LIN {X 0,Y 303.642,Z 314.333,A -85,B 0,C 180,E1 -15935.578,E2 -15935.578} C_VEL
LIN {X 0,Y 303.878,Z 309.685,A -85,B 0,C 180,E1 -15937.976,E2 -15937.976} C_VEL
LIN {X 0,Y 304.337,Z 303.514,A -85,B 0,C 180,E1 -15940.309,E2 -15940.309} C_VEL
LIN {X 0,Y 305.034,Z 296.766,A -85,B 0,C 180,E1 -15942.305,E2 -15942.305} C_VEL
LIN {X 0,Y 306.049,Z 288.388,A -85,B 0,C 180,E1 -15944.291,E2 -15944.291} C_VEL
LIN {X 0,Y 307.158,Z 279.773,A -85,B 0,C 180,E1 -15945.936,E2 -15945.936} C_VEL
LIN {X 0,Y 308.289,Z 269.101,A -85,B 0,C 180,E1 -15947.581,E2 -15947.581} C_VEL
LIN {X 0,Y 309.733,Z 258.568,A -85,B 0,C 180,E1 -15948.865,E2 -15948.865} C_VEL
LIN {X 0,Y 310.948,Z 246.911,A -85,B 0,C 180,E1 -15949.989,E2 -15949.989} C_VEL
LIN {X 0,Y 312.046,Z 234.79,A -85,B 0,C 180,E1 -15950.863,E2 -15950.863} C_VEL
LIN {X 0,Y 313.009,Z 221.635,A -85,B 0,C 180,E1 -15951.528,E2 -15951.528} C_VEL
LIN {X 0,Y 313.468,Z 208.98,A -85,B 0,C 180,E1 -15951.927,E2 -15951.927} C_VEL
LIN {X 0,Y 314.607,Z 149.7,A -85,B 0,C 180,E1 -15953.265,E2 -15953.265} C_VEL
LIN {X 0,Y 309.854,Z 113.898,A -85,B 0,C 180,E1 -15954.459,E2 -15954.459} C_VEL
LIN {X 0,Y 308.762,Z 106.65,A -85,B 0,C 180,E1 -15954.726,E2 -15954.726} C_VEL
LIN {X 0,Y 309.513,Z 100.612,A -85,B 0,C 180,E1 -15956.281,E2 -15956.281} C_VEL
LIN {X 0,Y 308.694,Z 94.627,A -85,B 0,C 180,E1 -15957.946,E2 -15957.946} C_VEL
LIN {X 0,Y 306.773,Z 85.34,A -85,B 0,C 180,E1 -15960.646,E2 -15960.646} C_VEL
LIN {X 0,Y 305.49,Z 79.435,A -85,B 0,C 180,E1 -15962.433,E2 -15962.433} C_VEL
LIN {X 0,Y 305.496,Z 79.432,A -85,B 0,C 180,E1 -15966.736,E2 -15966.736} C_VEL
LIN {X 0,Y 305.454,Z 79.435,A -85,B 0,C 180,E1 -15970.6,E2 -15970.6} C_VEL
LIN {X 0,Y 305.424,Z 79.442,A -85,B 0,C 180,E1 -15973.655,E2 -15973.655} C_VEL
LIN {X 0,Y 305.454,Z 79.438,A -85,B 0,C 180,E1 -15977.414,E2 -15977.414} C_VEL
LIN {X 0,Y 305.475,Z 79.428,A -85,B 0,C 180,E1 -15981.597,E2 -15981.597} C_VEL
LIN {X 0,Y 305.461,Z 79.435,A -85,B 0,C 180,E1 -15984.887,E2 -15984.887} C_VEL
LIN {X 0,Y 305.451,Z 79.435,A -85,B 0,C 180,E1 -15988.355,E2 -15988.355} C_VEL
LIN {X 0,Y 305.519,Z 79.429,A -85,B 0,C 180,E1 -15991.114,E2 -15991.114} C_VEL
LIN {X 0,Y 305.57,Z 79.417,A -85,B 0,C 180,E1 -15994.088,E2 -15994.088} C_VEL
LIN {X 0,Y 305.5,Z 79.429,A -85,B 0,C 180,E1 -15998.403,E2 -15998.403} C_VEL
LIN {X 0,Y 305.589,Z 79.417,A -85,B 0,C 180,E1 -16001.218,E2 -16001.218} C_VEL
LIN {X 0,Y 305.648,Z 79.408,A -85,B 0,C 180,E1 -16005.349,E2 -16005.349} C_VEL
LIN {X 0,Y 305.635,Z 79.409,A -85,B 0,C 180,E1 -16009.4,E2 -16009.4} C_VEL
LIN {X 0,Y 305.796,Z 79.394,A -85,B 0,C 180,E1 -16012.074,E2 -16012.074} C_VEL
LIN {X 0,Y 305.682,Z 79.404,A -85,B 0,C 180,E1 -16014.724,E2 -16014.724} C_VEL
LIN {X 0,Y 305.953,Z 79.372,A -85,B 0,C 180,E1 -16018.684,E2 -16018.684} C_VEL
LIN {X 0,Y 305.953,Z 79.372,A -85,B 0,C 180,E1 -16021.317,E2 -16021.317} C_VEL
LIN {X 0,Y 305.672,Z 79.402,A -85,B 0,C 180,E1 -16025.277,E2 -16025.277} C_VEL
LIN {X 0,Y 305.764,Z 79.399,A -85,B 0,C 180,E1 -16027.927,E2 -16027.927} C_VEL
LIN {X 0,Y 305.598,Z 79.414,A -85,B 0,C 180,E1 -16031.946,E2 -16031.946} C_VEL
LIN {X 0,Y 305.637,Z 79.409,A -85,B 0,C 180,E1 -16035.035,E2 -16035.035} C_VEL
LIN {X 0,Y 305.576,Z 79.42,A -85,B 0,C 180,E1 -16039.445,E2 -16039.445} C_VEL
LIN {X 0,Y 305.491,Z 79.428,A -85,B 0,C 180,E1 -16043.042,E2 -16043.042} C_VEL
LIN {X 0,Y 305.526,Z 79.424,A -85,B 0,C 180,E1 -16046.219,E2 -16046.219} C_VEL
LIN {X 0,Y 305.489,Z 79.433,A -85,B 0,C 180,E1 -16049.048,E2 -16049.048} C_VEL
LIN {X 0,Y 305.442,Z 79.435,A -85,B 0,C 180,E1 -16051.953,E2 -16051.953} C_VEL
LIN {X 0,Y 305.462,Z 79.437,A -85,B 0,C 180,E1 -16055.114,E2 -16055.114} C_VEL
LIN {X 0,Y 305.434,Z 79.438,A -85,B 0,C 180,E1 -16058.526,E2 -16058.526} C_VEL
LIN {X 0,Y 305.436,Z 79.44,A -85,B 0,C 180,E1 -16062.582,E2 -16062.582} C_VEL
LIN {X 0,Y 305.424,Z 79.441,A -85,B 0,C 180,E1 -16066.345,E2 -16066.345} C_VEL
LIN {X 0,Y 305.459,Z 79.434,A -85,B 0,C 180,E1 -16069.893,E2 -16069.893} C_VEL
LIN {X 0,Y 305.465,Z 79.433,A -85,B 0,C 180,E1 -16073.637,E2 -16073.637} C_VEL
LIN {X 0,Y 305.467,Z 79.434,A -85,B 0,C 180,E1 -16076.484,E2 -16076.484} C_VEL
LIN {X 0,Y 305.433,Z 79.437,A -85,B 0,C 180,E1 -16079.588,E2 -16079.588} C_VEL
LIN {X 0,Y 305.455,Z 79.436,A -85,B 0,C 180,E1 -16082.603,E2 -16082.603} C_VEL
LIN {X 0,Y 305.461,Z 79.435,A -85,B 0,C 180,E1 -16085.535,E2 -16085.535} C_VEL
LIN {X 0,Y 305.515,Z 79.431,A -85,B 0,C 180,E1 -16089.815,E2 -16089.815} C_VEL
LIN {X 0,Y 305.651,Z 79.555,A -85,B 0,C 180,E1 -16091.396,E2 -16091.396} C_VEL
LIN {X 0,Y 306.172,Z 82.09,A -85,B 0,C 180,E1 -16092.18,E2 -16092.18} C_VEL
LIN {X 0,Y 314.171,Z 104.116,A -85,B 0,C 180,E1 -16093.31,E2 -16093.31} C_VEL
LIN {X 0,Y 315.408,Z 109.173,A -85,B 0,C 180,E1 -16093.518,E2 -16093.518} C_VEL
LIN {X 0,Y 313.679,Z 189.055,A -85,B 0,C 180,E1 -16095.346,E2 -16095.346} C_VEL
LIN {X 0,Y 313.088,Z 202.338,A -85,B 0,C 180,E1 -16095.912,E2 -16095.912} C_VEL
LIN {X 0,Y 312.343,Z 214.286,A -85,B 0,C 180,E1 -16096.666,E2 -16096.666} C_VEL
LIN {X 0,Y 311.528,Z 225.57,A -85,B 0,C 180,E1 -16097.625,E2 -16097.625} C_VEL
LIN {X 0,Y 310.283,Z 237.207,A -85,B 0,C 180,E1 -16098.9,E2 -16098.9} C_VEL
LIN {X 0,Y 309.036,Z 247.649,A -85,B 0,C 180,E1 -16100.345,E2 -16100.345} C_VEL
LIN {X 0,Y 307.882,Z 256.196,A -85,B 0,C 180,E1 -16101.798,E2 -16101.798} C_VEL
LIN {X 0,Y 306.867,Z 264.064,A -85,B 0,C 180,E1 -16103.425,E2 -16103.425} C_VEL
LIN {X 0,Y 305.788,Z 271.78,A -85,B 0,C 180,E1 -16105.386,E2 -16105.386} C_VEL
LIN {X 0,Y 305.065,Z 277.948,A -85,B 0,C 180,E1 -16107.36,E2 -16107.36} C_VEL
LIN {X 0,Y 304.464,Z 282.865,A -85,B 0,C 180,E1 -16109.339,E2 -16109.339} C_VEL
LIN {X 0,Y 304.148,Z 286.666,A -85,B 0,C 180,E1 -16111.324,E2 -16111.324} C_VEL
LIN {X 0,Y 303.886,Z 288.636,A -85,B 0,C 180,E1 -16112.652,E2 -16112.652} C_VEL
LIN {X 0,Y 303.852,Z 290.188,A -85,B 0,C 180,E1 -16113.979,E2 -16113.979} C_VEL
LIN {X 0,Y 303.867,Z 291.727,A -85,B 0,C 180,E1 -16115.991,E2 -16115.991} C_VEL
LIN {X 0,Y 303.757,Z 292.363,A -85,B 0,C 180,E1 -16117.98,E2 -16117.98} C_VEL
LIN {X 0,Y 303.781,Z 292.317,A -85,B 0,C 180,E1 -16119.32,E2 -16119.32} C_VEL
LIN {X 0,Y 303.861,Z 291.854,A -85,B 0,C 180,E1 -16120.663,E2 -16120.663} C_VEL
LIN {X 0,Y 304.117,Z 290.967,A -85,B 0,C 180,E1 -16122.005,E2 -16122.005} C_VEL
LIN {X 0,Y 304.786,Z 288.35,A -85,B 0,C 180,E1 -16124.423,E2 -16124.423} C_VEL
LIN {X 0,Y 305.573,Z 284.582,A -85,B 0,C 180,E1 -16126.708,E2 -16126.708} C_VEL
LIN {X 0,Y 306.602,Z 280.053,A -85,B 0,C 180,E1 -16128.718,E2 -16128.718} C_VEL
LIN {X 0,Y 307.928,Z 273.826,A -85,B 0,C 180,E1 -16130.852,E2 -16130.852} C_VEL
LIN {X 0,Y 309.428,Z 266.966,A -85,B 0,C 180,E1 -16132.714,E2 -16132.714} C_VEL
LIN {X 0,Y 311.294,Z 257.875,A -85,B 0,C 180,E1 -16134.688,E2 -16134.688} C_VEL
LIN {X 0,Y 313.036,Z 248.077,A -85,B 0,C 180,E1 -16136.376,E2 -16136.376} C_VEL
LIN {X 0,Y 314.749,Z 237.818,A -85,B 0,C 180,E1 -16137.783,E2 -16137.783} C_VEL
LIN {X 0,Y 316.501,Z 225.991,A -85,B 0,C 180,E1 -16139.062,E2 -16139.062} C_VEL
LIN {X 0,Y 317.895,Z 214.405,A -85,B 0,C 180,E1 -16140.013,E2 -16140.013} C_VEL
LIN {X 0,Y 318.974,Z 201.792,A -85,B 0,C 180,E1 -16140.782,E2 -16140.782} C_VEL
LIN {X 0,Y 319.8,Z 188.955,A -85,B 0,C 180,E1 -16141.299,E2 -16141.299} C_VEL
LIN {X 0,Y 321.712,Z 116.244,A -85,B 0,C 180,E1 -16142.959,E2 -16142.959} C_VEL
LIN {X 0,Y 314.092,Z 98.688,A -85,B 0,C 180,E1 -16144.191,E2 -16144.191} C_VEL
LIN {X 0,Y 307.154,Z 84.745,A -85,B 0,C 180,E1 -16145.326,E2 -16145.326} C_VEL
LIN {X 0,Y 306.212,Z 82.518,A -85,B 0,C 180,E1 -16145.534,E2 -16145.534} C_VEL
LIN {X 0,Y 305.477,Z 79.43,A -85,B 0,C 180,E1 -16146.74,E2 -16146.74} C_VEL
LIN {X 0,Y 305.438,Z 79.432,A -85,B 0,C 180,E1 -16147.526,E2 -16147.526} C_VEL
LIN {X 0,Y 304.776,Z 79.521,A -85,B 0,C 180,E1 -16148.626,E2 -16148.626} C_VEL
LIN {X 0,Y 301.946,Z 79.88,A -85,B 0,C 180,E1 -16150.419,E2 -16150.419} C_VEL
LIN {X 0,Y 299.525,Z 80.183,A -85,B 0,C 180,E1 -16151.872,E2 -16151.872} C_VEL
LIN {X 0,Y 298.454,Z 80.309,A -85,B 0,C 180,E1 -16152.998,E2 -16152.998} C_VEL
LIN {X 0,Y 298.351,Z 80.315,A -85,B 0,C 180,E1 -16153.379,E2 -16153.379} C_VEL
LIN {X 0,Y 298.373,Z 80.318,A -85,B 0,C 180,E1 -16156.915,E2 -16156.915} C_VEL
LIN {X 0,Y 298.388,Z 80.313,A -85,B 0,C 180,E1 -16161.011,E2 -16161.011} C_VEL
LIN {X 0,Y 298.407,Z 80.31,A -85,B 0,C 180,E1 -16163.928,E2 -16163.928} C_VEL
LIN {X 0,Y 298.395,Z 80.314,A -85,B 0,C 180,E1 -16167.199,E2 -16167.199} C_VEL
LIN {X 0,Y 298.409,Z 80.307,A -85,B 0,C 180,E1 -16171.898,E2 -16171.898} C_VEL
LIN {X 0,Y 298.441,Z 80.312,A -85,B 0,C 180,E1 -16174.92,E2 -16174.92} C_VEL
LIN {X 0,Y 298.407,Z 80.305,A -85,B 0,C 180,E1 -16177.862,E2 -16177.862} C_VEL
LIN {X 0,Y 298.511,Z 80.298,A -85,B 0,C 180,E1 -16180.755,E2 -16180.755} C_VEL
LIN {X 0,Y 298.589,Z 80.293,A -85,B 0,C 180,E1 -16184.994,E2 -16184.994} C_VEL
LIN {X 0,Y 298.586,Z 80.285,A -85,B 0,C 180,E1 -16189.146,E2 -16189.146} C_VEL
LIN {X 0,Y 298.7,Z 80.277,A -85,B 0,C 180,E1 -16191.884,E2 -16191.884} C_VEL
LIN {X 0,Y 298.633,Z 80.274,A -85,B 0,C 180,E1 -16194.598,E2 -16194.598} C_VEL
LIN {X 0,Y 298.907,Z 80.242,A -85,B 0,C 180,E1 -16198.652,E2 -16198.652} C_VEL
LIN {X 0,Y 298.916,Z 80.244,A -85,B 0,C 180,E1 -16201.347,E2 -16201.347} C_VEL
LIN {X 0,Y 298.738,Z 80.261,A -85,B 0,C 180,E1 -16206.755,E2 -16206.755} C_VEL
LIN {X 0,Y 298.629,Z 80.286,A -85,B 0,C 180,E1 -16209.482,E2 -16209.482} C_VEL
LIN {X 0,Y 298.548,Z 80.292,A -85,B 0,C 180,E1 -16213.615,E2 -16213.615} C_VEL
LIN {X 0,Y 298.489,Z 80.293,A -85,B 0,C 180,E1 -16216.412,E2 -16216.412} C_VEL
LIN {X 0,Y 298.501,Z 80.303,A -85,B 0,C 180,E1 -16219.647,E2 -16219.647} C_VEL
LIN {X 0,Y 298.46,Z 80.304,A -85,B 0,C 180,E1 -16223.597,E2 -16223.597} C_VEL
LIN {X 0,Y 298.492,Z 80.295,A -85,B 0,C 180,E1 -16226.574,E2 -16226.574} C_VEL
LIN {X 0,Y 298.419,Z 80.311,A -85,B 0,C 180,E1 -16229.641,E2 -16229.641} C_VEL
LIN {X 0,Y 298.397,Z 80.316,A -85,B 0,C 180,E1 -16232.8,E2 -16232.8} C_VEL
LIN {X 0,Y 298.449,Z 80.281,A -85,B 0,C 180,E1 -16236.807,E2 -16236.807} C_VEL
LIN {X 0,Y 298.411,Z 80.314,A -85,B 0,C 180,E1 -16239.486,E2 -16239.486} C_VEL
LIN {X 0,Y 298.4,Z 80.315,A -85,B 0,C 180,E1 -16243.103,E2 -16243.103} C_VEL
LIN {X 0,Y 298.405,Z 80.312,A -85,B 0,C 180,E1 -16246.92,E2 -16246.92} C_VEL
LIN {X 0,Y 298.406,Z 80.311,A -85,B 0,C 180,E1 -16251.006,E2 -16251.006} C_VEL
LIN {X 0,Y 298.421,Z 80.369,A -85,B 0,C 180,E1 -16252.844,E2 -16252.844} C_VEL
LIN {X 0,Y 301.194,Z 91.103,A -85,B 0,C 180,E1 -16256.622,E2 -16256.622} C_VEL
LIN {X 0,Y 303.877,Z 103.194,A -85,B 0,C 180,E1 -16260.563,E2 -16260.563} C_VEL
LIN {X 0,Y 304.366,Z 105.671,A -85,B 0,C 180,E1 -16261.335,E2 -16261.335} C_VEL
LIN {X 0,Y 307.278,Z 113.342,A -85,B 0,C 180,E1 -16261.877,E2 -16261.877} C_VEL
LIN {X 0,Y 312.669,Z 141.354,A -85,B 0,C 180,E1 -16263.189,E2 -16263.189} C_VEL
LIN {X 0,Y 314.565,Z 154.061,A -85,B 0,C 180,E1 -16263.709,E2 -16263.709} C_VEL
LIN {X 0,Y 312.73,Z 215.019,A -85,B 0,C 180,E1 -16265.123,E2 -16265.123} C_VEL
LIN {X 0,Y 311.67,Z 228.866,A -85,B 0,C 180,E1 -16265.699,E2 -16265.699} C_VEL
LIN {X 0,Y 310.181,Z 241.295,A -85,B 0,C 180,E1 -16266.462,E2 -16266.462} C_VEL
LIN {X 0,Y 308.6,Z 252.386,A -85,B 0,C 180,E1 -16267.399,E2 -16267.399} C_VEL
LIN {X 0,Y 306.694,Z 263.941,A -85,B 0,C 180,E1 -16268.667,E2 -16268.667} C_VEL
LIN {X 0,Y 304.7,Z 274.36,A -85,B 0,C 180,E1 -16270.11,E2 -16270.11} C_VEL
LIN {X 0,Y 302.78,Z 283.763,A -85,B 0,C 180,E1 -16271.738,E2 -16271.738} C_VEL
LIN {X 0,Y 300.962,Z 292.85,A -85,B 0,C 180,E1 -16273.726,E2 -16273.726} C_VEL
LIN {X 0,Y 299.458,Z 300.197,A -85,B 0,C 180,E1 -16275.733,E2 -16275.733} C_VEL
LIN {X 0,Y 298.128,Z 306.106,A -85,B 0,C 180,E1 -16277.75,E2 -16277.75} C_VEL
LIN {X 0,Y 297.363,Z 310.791,A -85,B 0,C 180,E1 -16279.789,E2 -16279.789} C_VEL
LIN {X 0,Y 296.856,Z 314.38,A -85,B 0,C 180,E1 -16281.833,E2 -16281.833} C_VEL
LIN {X 0,Y 296.649,Z 316.232,A -85,B 0,C 180,E1 -16283.197,E2 -16283.197} C_VEL
LIN {X 0,Y 296.566,Z 318.639,A -85,B 0,C 180,E1 -16285.923,E2 -16285.923} C_VEL
LIN {X 0,Y 296.578,Z 319.259,A -85,B 0,C 180,E1 -16287.283,E2 -16287.283} C_VEL
LIN {X 0,Y 296.597,Z 319.477,A -85,B 0,C 180,E1 -16288.642,E2 -16288.642} C_VEL
LIN {X 0,Y 296.672,Z 319.265,A -85,B 0,C 180,E1 -16290,E2 -16290} C_VEL
LIN {X 0,Y 296.614,Z 318.655,A -85,B 0,C 180,E1 -16291.357,E2 -16291.357} C_VEL
LIN {X 0,Y 296.612,Z 317.653,A -85,B 0,C 180,E1 -16292.716,E2 -16292.716} C_VEL
LIN {X 0,Y 296.608,Z 316.234,A -85,B 0,C 180,E1 -16294.076,E2 -16294.076} C_VEL
LIN {X 0,Y 296.57,Z 313.254,A -85,B 0,C 180,E1 -16296.121,E2 -16296.121} C_VEL
LIN {X 0,Y 296.822,Z 309.219,A -85,B 0,C 180,E1 -16298.167,E2 -16298.167} C_VEL
LIN {X 0,Y 297.317,Z 302.992,A -85,B 0,C 180,E1 -16300.556,E2 -16300.556} C_VEL
LIN {X 0,Y 298.073,Z 296.199,A -85,B 0,C 180,E1 -16302.597,E2 -16302.597} C_VEL
LIN {X 0,Y 299.144,Z 287.762,A -85,B 0,C 180,E1 -16304.628,E2 -16304.628} C_VEL
LIN {X 0,Y 300.236,Z 279.054,A -85,B 0,C 180,E1 -16306.313,E2 -16306.313} C_VEL
LIN {X 0,Y 301.318,Z 269.493,A -85,B 0,C 180,E1 -16307.826,E2 -16307.826} C_VEL
LIN {X 0,Y 302.989,Z 257.676,A -85,B 0,C 180,E1 -16309.301,E2 -16309.301} C_VEL
LIN {X 0,Y 304.247,Z 245.794,A -85,B 0,C 180,E1 -16310.449,E2 -16310.449} C_VEL
LIN {X 0,Y 305.395,Z 233.429,A -85,B 0,C 180,E1 -16311.339,E2 -16311.339} C_VEL
LIN {X 0,Y 306.33,Z 220.772,A -85,B 0,C 180,E1 -16311.978,E2 -16311.978} C_VEL
LIN {X 0,Y 306.817,Z 207.603,A -85,B 0,C 180,E1 -16312.384,E2 -16312.384} C_VEL
LIN {X 0,Y 307.946,Z 150.508,A -85,B 0,C 180,E1 -16313.7,E2 -16313.7} C_VEL
LIN {X 0,Y 303.523,Z 116.739,A -85,B 0,C 180,E1 -16314.855,E2 -16314.855} C_VEL
LIN {X 0,Y 301.95,Z 106.265,A -85,B 0,C 180,E1 -16315.262,E2 -16315.262} C_VEL
LIN {X 0,Y 302.573,Z 101.353,A -85,B 0,C 180,E1 -16316.559,E2 -16316.559} C_VEL
LIN {X 0,Y 301.205,Z 93.039,A -85,B 0,C 180,E1 -16318.957,E2 -16318.957} C_VEL
LIN {X 0,Y 298.456,Z 80.312,A -85,B 0,C 180,E1 -16322.842,E2 -16322.842} C_VEL
LIN {X 0,Y 298.464,Z 80.309,A -85,B 0,C 180,E1 -16326.812,E2 -16326.812} C_VEL
LIN {X 0,Y 298.386,Z 80.316,A -85,B 0,C 180,E1 -16331.088,E2 -16331.088} C_VEL
LIN {X 0,Y 298.397,Z 80.315,A -85,B 0,C 180,E1 -16333.103,E2 -16333.103} C_VEL
LIN {X 0,Y 298.402,Z 80.314,A -85,B 0,C 180,E1 -16336.921,E2 -16336.921} C_VEL
LIN {X 0,Y 298.403,Z 80.307,A -85,B 0,C 180,E1 -16341.006,E2 -16341.006} C_VEL
LIN {X 0,Y 298.417,Z 80.31,A -85,B 0,C 180,E1 -16343.93,E2 -16343.93} C_VEL
LIN {X 0,Y 298.394,Z 80.313,A -85,B 0,C 180,E1 -16347.983,E2 -16347.983} C_VEL
LIN {X 0,Y 298.462,Z 80.304,A -85,B 0,C 180,E1 -16351.904,E2 -16351.904} C_VEL
LIN {X 0,Y 298.485,Z 80.305,A -85,B 0,C 180,E1 -16354.924,E2 -16354.924} C_VEL
LIN {X 0,Y 298.449,Z 80.302,A -85,B 0,C 180,E1 -16359.315,E2 -16359.315} C_VEL
LIN {X 0,Y 298.537,Z 80.295,A -85,B 0,C 180,E1 -16362.18,E2 -16362.18} C_VEL
LIN {X 0,Y 298.592,Z 80.289,A -85,B 0,C 180,E1 -16364.995,E2 -16364.995} C_VEL
LIN {X 0,Y 298.591,Z 80.287,A -85,B 0,C 180,E1 -16369.147,E2 -16369.147} C_VEL
LIN {X 0,Y 298.74,Z 80.272,A -85,B 0,C 180,E1 -16371.886,E2 -16371.886} C_VEL
LIN {X 0,Y 298.653,Z 80.28,A -85,B 0,C 180,E1 -16374.599,E2 -16374.599} C_VEL
LIN {X 0,Y 298.919,Z 80.248,A -85,B 0,C 180,E1 -16378.653,E2 -16378.653} C_VEL
LIN {X 0,Y 298.919,Z 80.248,A -85,B 0,C 180,E1 -16381.348,E2 -16381.348} C_VEL
LIN {X 0,Y 298.716,Z 80.269,A -85,B 0,C 180,E1 -16386.515,E2 -16386.515} C_VEL
LIN {X 0,Y 298.625,Z 80.286,A -85,B 0,C 180,E1 -16389.483,E2 -16389.483} C_VEL
LIN {X 0,Y 298.552,Z 80.291,A -85,B 0,C 180,E1 -16393.616,E2 -16393.616} C_VEL
LIN {X 0,Y 298.549,Z 80.293,A -85,B 0,C 180,E1 -16396.409,E2 -16396.409} C_VEL
LIN {X 0,Y 298.511,Z 80.298,A -85,B 0,C 180,E1 -16399.655,E2 -16399.655} C_VEL
LIN {X 0,Y 298.458,Z 80.307,A -85,B 0,C 180,E1 -16403.598,E2 -16403.598} C_VEL
LIN {X 0,Y 298.485,Z 80.302,A -85,B 0,C 180,E1 -16406.575,E2 -16406.575} C_VEL
LIN {X 0,Y 298.417,Z 80.311,A -85,B 0,C 180,E1 -16409.642,E2 -16409.642} C_VEL
LIN {X 0,Y 298.395,Z 80.316,A -85,B 0,C 180,E1 -16412.801,E2 -16412.801} C_VEL
LIN {X 0,Y 298.442,Z 80.312,A -85,B 0,C 180,E1 -16416.807,E2 -16416.807} C_VEL
LIN {X 0,Y 298.348,Z 80.321,A -85,B 0,C 180,E1 -16421.08,E2 -16421.08} C_VEL
LIN {X 0,Y 298.355,Z 80.321,A -85,B 0,C 180,E1 -16425.035,E2 -16425.035} C_VEL
LIN {X 0,Y 298.378,Z 80.319,A -85,B 0,C 180,E1 -16428.738,E2 -16428.738} C_VEL
LIN {X 0,Y 298.401,Z 80.316,A -85,B 0,C 180,E1 -16432.24,E2 -16432.24} C_VEL
LIN {X 0,Y 298.41,Z 80.312,A -85,B 0,C 180,E1 -16435.582,E2 -16435.582} C_VEL
LIN {X 0,Y 298.379,Z 80.316,A -85,B 0,C 180,E1 -16438.79,E2 -16438.79} C_VEL
LIN {X 0,Y 298.413,Z 80.308,A -85,B 0,C 180,E1 -16441.9,E2 -16441.9} C_VEL
LIN {X 0,Y 298.426,Z 80.31,A -85,B 0,C 180,E1 -16444.919,E2 -16444.919} C_VEL
LIN {X 0,Y 298.442,Z 80.31,A -85,B 0,C 180,E1 -16449.315,E2 -16449.315} C_VEL
LIN {X 0,Y 298.61,Z 80.499,A -85,B 0,C 180,E1 -16451.029,E2 -16451.029} C_VEL
LIN {X 0,Y 298.99,Z 82.133,A -85,B 0,C 180,E1 -16451.596,E2 -16451.596} C_VEL
LIN {X 0,Y 307.413,Z 105.14,A -85,B 0,C 180,E1 -16452.845,E2 -16452.845} C_VEL
LIN {X 0,Y 308.835,Z 110.398,A -85,B 0,C 180,E1 -16453.079,E2 -16453.079} C_VEL
LIN {X 0,Y 306.98,Z 189.257,A -85,B 0,C 180,E1 -16454.913,E2 -16454.913} C_VEL
LIN {X 0,Y 306.406,Z 202.19,A -85,B 0,C 180,E1 -16455.471,E2 -16455.471} C_VEL
LIN {X 0,Y 305.592,Z 214.817,A -85,B 0,C 180,E1 -16456.281,E2 -16456.281} C_VEL
LIN {X 0,Y 304.632,Z 226.842,A -85,B 0,C 180,E1 -16457.34,E2 -16457.34} C_VEL
LIN {X 0,Y 303.367,Z 238.289,A -85,B 0,C 180,E1 -16458.644,E2 -16458.644} C_VEL
LIN {X 0,Y 302.079,Z 248.601,A -85,B 0,C 180,E1 -16460.121,E2 -16460.121} C_VEL
LIN {X 0,Y 300.895,Z 257.042,A -85,B 0,C 180,E1 -16461.606,E2 -16461.606} C_VEL
LIN {X 0,Y 299.851,Z 264.82,A -85,B 0,C 180,E1 -16463.27,E2 -16463.27} C_VEL
LIN {X 0,Y 298.744,Z 272.429,A -85,B 0,C 180,E1 -16465.277,E2 -16465.277} C_VEL
LIN {X 0,Y 298.015,Z 278.534,A -85,B 0,C 180,E1 -16467.297,E2 -16467.297} C_VEL
LIN {X 0,Y 297.382,Z 283.396,A -85,B 0,C 180,E1 -16469.323,E2 -16469.323} C_VEL
LIN {X 0,Y 297.04,Z 287.145,A -85,B 0,C 180,E1 -16471.356,E2 -16471.356} C_VEL
LIN {X 0,Y 296.798,Z 289.089,A -85,B 0,C 180,E1 -16472.715,E2 -16472.715} C_VEL
LIN {X 0,Y 296.78,Z 290.613,A -85,B 0,C 180,E1 -16474.074,E2 -16474.074} C_VEL
LIN {X 0,Y 296.785,Z 292.006,A -85,B 0,C 180,E1 -16475.963,E2 -16475.963} C_VEL
LIN {X 0,Y 296.665,Z 292.698,A -85,B 0,C 180,E1 -16478.172,E2 -16478.172} C_VEL
LIN {X 0,Y 296.71,Z 292.625,A -85,B 0,C 180,E1 -16479.544,E2 -16479.544} C_VEL
LIN {X 0,Y 296.807,Z 292.117,A -85,B 0,C 180,E1 -16480.92,E2 -16480.92} C_VEL
LIN {X 0,Y 297.094,Z 291.206,A -85,B 0,C 180,E1 -16482.293,E2 -16482.293} C_VEL
LIN {X 0,Y 297.765,Z 288.758,A -85,B 0,C 180,E1 -16484.599,E2 -16484.599} C_VEL
LIN {X 0,Y 298.664,Z 284.708,A -85,B 0,C 180,E1 -16487.107,E2 -16487.107} C_VEL
LIN {X 0,Y 299.776,Z 280.115,A -85,B 0,C 180,E1 -16489.161,E2 -16489.161} C_VEL
LIN {X 0,Y 301.355,Z 273.044,A -85,B 0,C 180,E1 -16491.575,E2 -16491.575} C_VEL
LIN {X 0,Y 303.097,Z 265.516,A -85,B 0,C 180,E1 -16493.577,E2 -16493.577} C_VEL
LIN {X 0,Y 304.755,Z 257.691,A -85,B 0,C 180,E1 -16495.254,E2 -16495.254} C_VEL
LIN {X 0,Y 306.554,Z 247.997,A -85,B 0,C 180,E1 -16496.937,E2 -16496.937} C_VEL
LIN {X 0,Y 308.383,Z 237.36,A -85,B 0,C 180,E1 -16498.408,E2 -16498.408} C_VEL
LIN {X 0,Y 309.976,Z 226.972,A -85,B 0,C 180,E1 -16499.547,E2 -16499.547} C_VEL
LIN {X 0,Y 311.535,Z 214.756,A -85,B 0,C 180,E1 -16500.577,E2 -16500.577} C_VEL
LIN {X 0,Y 312.634,Z 202.266,A -85,B 0,C 180,E1 -16501.356,E2 -16501.356} C_VEL
LIN {X 0,Y 313.514,Z 189.064,A -85,B 0,C 180,E1 -16501.896,E2 -16501.896} C_VEL
LIN {X 0,Y 315.447,Z 118.08,A -85,B 0,C 180,E1 -16503.547,E2 -16503.547} C_VEL
LIN {X 0,Y 308.063,Z 101.092,A -85,B 0,C 180,E1 -16504.785,E2 -16504.785} C_VEL
LIN {X 0,Y 300.454,Z 85.893,A -85,B 0,C 180,E1 -16506.081,E2 -16506.081} C_VEL
LIN {X 0,Y 299.054,Z 82.948,A -85,B 0,C 180,E1 -16506.354,E2 -16506.354} C_VEL
LIN {X 0,Y 298.399,Z 80.308,A -85,B 0,C 180,E1 -16507.426,E2 -16507.426} C_VEL
LIN {X 0,Y 298.35,Z 80.321,A -85,B 0,C 180,E1 -16511.268,E2 -16511.268} C_VEL
LIN {X 0,Y 298.351,Z 80.315,A -85,B 0,C 180,E1 -16513.379,E2 -16513.379} C_VEL
LIN {X 0,Y 297.64,Z 80.395,A -85,B 0,C 180,E1 -16514.506,E2 -16514.506} C_VEL
LIN {X 0,Y 294.787,Z 80.76,A -85,B 0,C 180,E1 -16516.341,E2 -16516.341} C_VEL
LIN {X 0,Y 292.399,Z 81.063,A -85,B 0,C 180,E1 -16517.83,E2 -16517.83} C_VEL
LIN {X 0,Y 291.383,Z 81.188,A -85,B 0,C 180,E1 -16518.983,E2 -16518.983} C_VEL
LIN {X 0,Y 291.302,Z 81.197,A -85,B 0,C 180,E1 -16519.373,E2 -16519.373} C_VEL
LIN {X 0,Y 291.388,Z 81.188,A -85,B 0,C 180,E1 -16522.916,E2 -16522.916} C_VEL
LIN {X 0,Y 291.346,Z 81.193,A -85,B 0,C 180,E1 -16526.301,E2 -16526.301} C_VEL
LIN {X 0,Y 291.341,Z 81.194,A -85,B 0,C 180,E1 -16530.277,E2 -16530.277} C_VEL
LIN {X 0,Y 291.361,Z 81.19,A -85,B 0,C 180,E1 -16534.266,E2 -16534.266} C_VEL
LIN {X 0,Y 291.368,Z 81.18,A -85,B 0,C 180,E1 -16537.298,E2 -16537.298} C_VEL
LIN {X 0,Y 291.462,Z 81.179,A -85,B 0,C 180,E1 -16540.27,E2 -16540.27} C_VEL
LIN {X 0,Y 291.501,Z 81.174,A -85,B 0,C 180,E1 -16544.665,E2 -16544.665} C_VEL
LIN {X 0,Y 291.532,Z 81.16,A -85,B 0,C 180,E1 -16548.88,E2 -16548.88} C_VEL
LIN {X 0,Y 291.654,Z 81.154,A -85,B 0,C 180,E1 -16551.687,E2 -16551.687} C_VEL
LIN {X 0,Y 291.602,Z 81.148,A -85,B 0,C 180,E1 -16554.467,E2 -16554.467} C_VEL
LIN {X 0,Y 291.874,Z 81.118,A -85,B 0,C 180,E1 -16558.62,E2 -16558.62} C_VEL
LIN {X 0,Y 291.882,Z 81.12,A -85,B 0,C 180,E1 -16561.379,E2 -16561.379} C_VEL
LIN {X 0,Y 291.69,Z 81.14,A -85,B 0,C 180,E1 -16566.919,E2 -16566.919} C_VEL
LIN {X 0,Y 291.571,Z 81.163,A -85,B 0,C 180,E1 -16569.714,E2 -16569.714} C_VEL
LIN {X 0,Y 291.518,Z 81.171,A -85,B 0,C 180,E1 -16573.95,E2 -16573.95} C_VEL
LIN {X 0,Y 291.451,Z 81.173,A -85,B 0,C 180,E1 -16578.269,E2 -16578.269} C_VEL
LIN {X 0,Y 291.376,Z 81.183,A -85,B 0,C 180,E1 -16581.211,E2 -16581.211} C_VEL
LIN {X 0,Y 291.403,Z 81.186,A -85,B 0,C 180,E1 -16584.205,E2 -16584.205} C_VEL
LIN {X 0,Y 291.423,Z 81.176,A -85,B 0,C 180,E1 -16587.271,E2 -16587.271} C_VEL
LIN {X 0,Y 291.337,Z 81.19,A -85,B 0,C 180,E1 -16590.437,E2 -16590.437} C_VEL
LIN {X 0,Y 291.347,Z 81.191,A -85,B 0,C 180,E1 -16593.698,E2 -16593.698} C_VEL
LIN {X 0,Y 291.383,Z 81.163,A -85,B 0,C 180,E1 -16597.255,E2 -16597.255} C_VEL
LIN {X 0,Y 291.336,Z 81.192,A -85,B 0,C 180,E1 -16600.642,E2 -16600.642} C_VEL
LIN {X 0,Y 291.292,Z 81.2,A -85,B 0,C 180,E1 -16604.401,E2 -16604.401} C_VEL
LIN {X 0,Y 291.328,Z 81.19,A -85,B 0,C 180,E1 -16608.404,E2 -16608.404} C_VEL
LIN {X 0,Y 291.396,Z 81.331,A -85,B 0,C 180,E1 -16612.126,E2 -16612.126} C_VEL
LIN {X 0,Y 293.717,Z 90.164,A -85,B 0,C 180,E1 -16615.369,E2 -16615.369} C_VEL
LIN {X 0,Y 295.964,Z 100.019,A -85,B 0,C 180,E1 -16618.744,E2 -16618.744} C_VEL
LIN {X 0,Y 297.139,Z 105.368,A -85,B 0,C 180,E1 -16620.485,E2 -16620.485} C_VEL
LIN {X 0,Y 301.287,Z 115.289,A -85,B 0,C 180,E1 -16621.251,E2 -16621.251} C_VEL
LIN {X 0,Y 306.1,Z 140.217,A -85,B 0,C 180,E1 -16622.464,E2 -16622.464} C_VEL
LIN {X 0,Y 308.319,Z 154.694,A -85,B 0,C 180,E1 -16623.084,E2 -16623.084} C_VEL
LIN {X 0,Y 306.469,Z 214.286,A -85,B 0,C 180,E1 -16624.488,E2 -16624.488} C_VEL
LIN {X 0,Y 305.463,Z 227.505,A -85,B 0,C 180,E1 -16625.036,E2 -16625.036} C_VEL
LIN {X 0,Y 303.877,Z 240.769,A -85,B 0,C 180,E1 -16625.853,E2 -16625.853} C_VEL
LIN {X 0,Y 302.089,Z 252.702,A -85,B 0,C 180,E1 -16626.884,E2 -16626.884} C_VEL
LIN {X 0,Y 300.104,Z 264.138,A -85,B 0,C 180,E1 -16628.175,E2 -16628.175} C_VEL
LIN {X 0,Y 298.025,Z 274.466,A -85,B 0,C 180,E1 -16629.645,E2 -16629.645} C_VEL
LIN {X 0,Y 296.037,Z 283.767,A -85,B 0,C 180,E1 -16631.307,E2 -16631.307} C_VEL
LIN {X 0,Y 294.15,Z 292.797,A -85,B 0,C 180,E1 -16633.338,E2 -16633.338} C_VEL
LIN {X 0,Y 292.573,Z 300.096,A -85,B 0,C 180,E1 -16635.39,E2 -16635.39} C_VEL
LIN {X 0,Y 291.16,Z 305.963,A -85,B 0,C 180,E1 -16637.453,E2 -16637.453} C_VEL
LIN {X 0,Y 290.344,Z 310.609,A -85,B 0,C 180,E1 -16639.54,E2 -16639.54} C_VEL
LIN {X 0,Y 289.817,Z 314.164,A -85,B 0,C 180,E1 -16641.633,E2 -16641.633} C_VEL
LIN {X 0,Y 289.575,Z 315.982,A -85,B 0,C 180,E1 -16643.03,E2 -16643.03} C_VEL
LIN {X 0,Y 289.464,Z 318.357,A -85,B 0,C 180,E1 -16645.823,E2 -16645.823} C_VEL
LIN {X 0,Y 289.503,Z 318.962,A -85,B 0,C 180,E1 -16647.217,E2 -16647.217} C_VEL
LIN {X 0,Y 289.512,Z 319.151,A -85,B 0,C 180,E1 -16648.609,E2 -16648.609} C_VEL
LIN {X 0,Y 289.582,Z 318.921,A -85,B 0,C 180,E1 -16650,E2 -16650} C_VEL
LIN {X 0,Y 289.53,Z 318.295,A -85,B 0,C 180,E1 -16651.391,E2 -16651.391} C_VEL
LIN {X 0,Y 289.536,Z 317.277,A -85,B 0,C 180,E1 -16652.782,E2 -16652.782} C_VEL
LIN {X 0,Y 289.519,Z 315.827,A -85,B 0,C 180,E1 -16654.176,E2 -16654.176} C_VEL
LIN {X 0,Y 289.489,Z 312.816,A -85,B 0,C 180,E1 -16656.272,E2 -16656.272} C_VEL
LIN {X 0,Y 289.758,Z 308.745,A -85,B 0,C 180,E1 -16658.367,E2 -16658.367} C_VEL
LIN {X 0,Y 290.293,Z 302.468,A -85,B 0,C 180,E1 -16660.814,E2 -16660.814} C_VEL
LIN {X 0,Y 291.107,Z 295.63,A -85,B 0,C 180,E1 -16662.904,E2 -16662.904} C_VEL
LIN {X 0,Y 292.258,Z 287.125,A -85,B 0,C 180,E1 -16664.981,E2 -16664.981} C_VEL
LIN {X 0,Y 293.361,Z 278.339,A -85,B 0,C 180,E1 -16666.707,E2 -16666.707} C_VEL
LIN {X 0,Y 294.567,Z 268.707,A -85,B 0,C 180,E1 -16668.249,E2 -16668.249} C_VEL
LIN {X 0,Y 296.076,Z 258.223,A -85,B 0,C 180,E1 -16669.59,E2 -16669.59} C_VEL
LIN {X 0,Y 297.364,Z 246.664,A -85,B 0,C 180,E1 -16670.763,E2 -16670.763} C_VEL
LIN {X 0,Y 298.535,Z 234.685,A -85,B 0,C 180,E1 -16671.673,E2 -16671.673} C_VEL
LIN {X 0,Y 299.578,Z 221.754,A -85,B 0,C 180,E1 -16672.363,E2 -16672.363} C_VEL
LIN {X 0,Y 300.059,Z 209.657,A -85,B 0,C 180,E1 -16672.78,E2 -16672.78} C_VEL
LIN {X 0,Y 301.237,Z 150.623,A -85,B 0,C 180,E1 -16674.176,E2 -16674.176} C_VEL
LIN {X 0,Y 296.791,Z 116.705,A -85,B 0,C 180,E1 -16675.373,E2 -16675.373} C_VEL
LIN {X 0,Y 295.208,Z 105.988,A -85,B 0,C 180,E1 -16675.79,E2 -16675.79} C_VEL
LIN {X 0,Y 295.592,Z 102.083,A -85,B 0,C 180,E1 -16676.855,E2 -16676.855} C_VEL
LIN {X 0,Y 293.845,Z 92.371,A -85,B 0,C 180,E1 -16679.754,E2 -16679.754} C_VEL
LIN {X 0,Y 291.387,Z 81.194,A -85,B 0,C 180,E1 -16683.285,E2 -16683.285} C_VEL
LIN {X 0,Y 291.394,Z 81.191,A -85,B 0,C 180,E1 -16687.259,E2 -16687.259} C_VEL
LIN {X 0,Y 291.333,Z 81.194,A -85,B 0,C 180,E1 -16690.642,E2 -16690.642} C_VEL
LIN {X 0,Y 291.289,Z 81.199,A -85,B 0,C 180,E1 -16694.402,E2 -16694.402} C_VEL
LIN {X 0,Y 291.325,Z 81.194,A -85,B 0,C 180,E1 -16698.404,E2 -16698.404} C_VEL
LIN {X 0,Y 291.351,Z 81.184,A -85,B 0,C 180,E1 -16701.158,E2 -16701.158} C_VEL
LIN {X 0,Y 291.36,Z 81.189,A -85,B 0,C 180,E1 -16704.626,E2 -16704.626} C_VEL
LIN {X 0,Y 291.371,Z 81.188,A -85,B 0,C 180,E1 -16707.951,E2 -16707.951} C_VEL
LIN {X 0,Y 291.381,Z 81.189,A -85,B 0,C 180,E1 -16711.158,E2 -16711.158} C_VEL
LIN {X 0,Y 291.415,Z 81.18,A -85,B 0,C 180,E1 -16714.272,E2 -16714.272} C_VEL
LIN {X 0,Y 291.381,Z 81.187,A -85,B 0,C 180,E1 -16717.3,E2 -16717.3} C_VEL
LIN {X 0,Y 291.457,Z 81.173,A -85,B 0,C 180,E1 -16720.27,E2 -16720.27} C_VEL
LIN {X 0,Y 291.554,Z 81.168,A -85,B 0,C 180,E1 -16724.624,E2 -16724.624} C_VEL
LIN {X 0,Y 291.535,Z 81.167,A -85,B 0,C 180,E1 -16728.881,E2 -16728.881} C_VEL
LIN {X 0,Y 291.687,Z 81.149,A -85,B 0,C 180,E1 -16731.688,E2 -16731.688} C_VEL
LIN {X 0,Y 291.624,Z 81.156,A -85,B 0,C 180,E1 -16734.468,E2 -16734.468} C_VEL
LIN {X 0,Y 291.886,Z 81.124,A -85,B 0,C 180,E1 -16738.621,E2 -16738.621} C_VEL
LIN {X 0,Y 291.886,Z 81.124,A -85,B 0,C 180,E1 -16741.38,E2 -16741.38} C_VEL
LIN {X 0,Y 291.699,Z 81.145,A -85,B 0,C 180,E1 -16746.919,E2 -16746.919} C_VEL
LIN {X 0,Y 291.568,Z 81.167,A -85,B 0,C 180,E1 -16749.714,E2 -16749.714} C_VEL
LIN {X 0,Y 291.522,Z 81.168,A -85,B 0,C 180,E1 -16753.951,E2 -16753.951} C_VEL
LIN {X 0,Y 291.487,Z 81.173,A -85,B 0,C 180,E1 -16756.818,E2 -16756.818} C_VEL
LIN {X 0,Y 291.451,Z 81.175,A -85,B 0,C 180,E1 -16759.875,E2 -16759.875} C_VEL
LIN {X 0,Y 291.399,Z 81.184,A -85,B 0,C 180,E1 -16764.206,E2 -16764.206} C_VEL
LIN {X 0,Y 291.419,Z 81.185,A -85,B 0,C 180,E1 -16767.272,E2 -16767.272} C_VEL
LIN {X 0,Y 291.335,Z 81.193,A -85,B 0,C 180,E1 -16770.438,E2 -16770.438} C_VEL
LIN {X 0,Y 291.345,Z 81.192,A -85,B 0,C 180,E1 -16773.699,E2 -16773.699} C_VEL
LIN {X 0,Y 291.369,Z 81.19,A -85,B 0,C 180,E1 -16777.253,E2 -16777.253} C_VEL
LIN {X 0,Y 291.3,Z 81.201,A -85,B 0,C 180,E1 -16780.649,E2 -16780.649} C_VEL
LIN {X 0,Y 291.282,Z 81.202,A -85,B 0,C 180,E1 -16784.404,E2 -16784.404} C_VEL
LIN {X 0,Y 291.322,Z 81.197,A -85,B 0,C 180,E1 -16788.406,E2 -16788.406} C_VEL
LIN {X 0,Y 291.345,Z 81.192,A -85,B 0,C 180,E1 -16791.158,E2 -16791.158} C_VEL
LIN {X 0,Y 291.357,Z 81.193,A -85,B 0,C 180,E1 -16794.626,E2 -16794.626} C_VEL
LIN {X 0,Y 291.368,Z 81.189,A -85,B 0,C 180,E1 -16797.951,E2 -16797.951} C_VEL
LIN {X 0,Y 291.345,Z 81.185,A -85,B 0,C 180,E1 -16801.155,E2 -16801.155} C_VEL
LIN {X 0,Y 291.351,Z 81.194,A -85,B 0,C 180,E1 -16804.266,E2 -16804.266} C_VEL
LIN {X 0,Y 291.366,Z 81.191,A -85,B 0,C 180,E1 -16807.299,E2 -16807.299} C_VEL
LIN {X 0,Y 291.525,Z 81.31,A -85,B 0,C 180,E1 -16810.596,E2 -16810.596} C_VEL
LIN {X 0,Y 291.866,Z 82.752,A -85,B 0,C 180,E1 -16811.04,E2 -16811.04} C_VEL
LIN {X 0,Y 299.789,Z 103.698,A -85,B 0,C 180,E1 -16812.228,E2 -16812.228} C_VEL
LIN {X 0,Y 302.203,Z 111.477,A -85,B 0,C 180,E1 -16812.611,E2 -16812.611} C_VEL
LIN {X 0,Y 300.293,Z 189.794,A -85,B 0,C 180,E1 -16814.474,E2 -16814.474} C_VEL
LIN {X 0,Y 299.683,Z 202.798,A -85,B 0,C 180,E1 -16815.051,E2 -16815.051} C_VEL
LIN {X 0,Y 298.85,Z 215.349,A -85,B 0,C 180,E1 -16815.878,E2 -16815.878} C_VEL
LIN {X 0,Y 297.927,Z 226.525,A -85,B 0,C 180,E1 -16816.877,E2 -16816.877} C_VEL
LIN {X 0,Y 296.62,Z 238.089,A -85,B 0,C 180,E1 -16818.208,E2 -16818.208} C_VEL
LIN {X 0,Y 295.286,Z 248.489,A -85,B 0,C 180,E1 -16819.718,E2 -16819.718} C_VEL
LIN {X 0,Y 293.911,Z 257.877,A -85,B 0,C 180,E1 -16821.405,E2 -16821.405} C_VEL
LIN {X 0,Y 292.634,Z 266.902,A -85,B 0,C 180,E1 -16823.45,E2 -16823.45} C_VEL
LIN {X 0,Y 291.54,Z 274.187,A -85,B 0,C 180,E1 -16825.507,E2 -16825.507} C_VEL
LIN {X 0,Y 290.721,Z 280.866,A -85,B 0,C 180,E1 -16827.922,E2 -16827.922} C_VEL
LIN {X 0,Y 290.195,Z 285.286,A -85,B 0,C 180,E1 -16830,E2 -16830} C_VEL
LIN {X 0,Y 289.933,Z 287.624,A -85,B 0,C 180,E1 -16831.389,E2 -16831.389} C_VEL
LIN {X 0,Y 289.713,Z 289.541,A -85,B 0,C 180,E1 -16832.781,E2 -16832.781} C_VEL
LIN {X 0,Y 289.687,Z 291.028,A -85,B 0,C 180,E1 -16834.174,E2 -16834.174} C_VEL
LIN {X 0,Y 289.687,Z 292.267,A -85,B 0,C 180,E1 -16835.902,E2 -16835.902} C_VEL
LIN {X 0,Y 289.571,Z 293.033,A -85,B 0,C 180,E1 -16838.374,E2 -16838.374} C_VEL
LIN {X 0,Y 289.627,Z 292.922,A -85,B 0,C 180,E1 -16839.78,E2 -16839.78} C_VEL
LIN {X 0,Y 290.085,Z 291.445,A -85,B 0,C 180,E1 -16842.595,E2 -16842.595} C_VEL
LIN {X 0,Y 290.733,Z 289.181,A -85,B 0,C 180,E1 -16844.772,E2 -16844.772} C_VEL
LIN {X 0,Y 291.453,Z 286.096,A -85,B 0,C 180,E1 -16846.82,E2 -16846.82} C_VEL
LIN {X 0,Y 292.539,Z 281.835,A -85,B 0,C 180,E1 -16848.925,E2 -16848.925} C_VEL
LIN {X 0,Y 293.982,Z 275.86,A -85,B 0,C 180,E1 -16851.195,E2 -16851.195} C_VEL
LIN {X 0,Y 295.521,Z 269.481,A -85,B 0,C 180,E1 -16853.104,E2 -16853.104} C_VEL
LIN {X 0,Y 297.142,Z 262.424,A -85,B 0,C 180,E1 -16854.824,E2 -16854.824} C_VEL
LIN {X 0,Y 298.973,Z 253.866,A -85,B 0,C 180,E1 -16856.529,E2 -16856.529} C_VEL
LIN {X 0,Y 300.907,Z 243.227,A -85,B 0,C 180,E1 -16858.227,E2 -16858.227} C_VEL
LIN {X 0,Y 302.787,Z 232.645,A -85,B 0,C 180,E1 -16859.554,E2 -16859.554} C_VEL
LIN {X 0,Y 304.489,Z 221.125,A -85,B 0,C 180,E1 -16860.687,E2 -16860.687} C_VEL
LIN {X 0,Y 305.761,Z 208.891,A -85,B 0,C 180,E1 -16861.601,E2 -16861.601} C_VEL
LIN {X 0,Y 306.884,Z 195.956,A -85,B 0,C 180,E1 -16862.269,E2 -16862.269} C_VEL
LIN {X 0,Y 307.486,Z 183.055,A -85,B 0,C 180,E1 -16862.683,E2 -16862.683} C_VEL
LIN {X 0,Y 309.291,Z 120.035,A -85,B 0,C 180,E1 -16864.148,E2 -16864.148} C_VEL
LIN {X 0,Y 301.715,Z 102.836,A -85,B 0,C 180,E1 -16865.464,E2 -16865.464} C_VEL
LIN {X 0,Y 295.13,Z 89.729,A -85,B 0,C 180,E1 -16866.627,E2 -16866.627} C_VEL
LIN {X 0,Y 291.914,Z 83.314,A -85,B 0,C 180,E1 -16867.245,E2 -16867.245} C_VEL
LIN {X 0,Y 291.346,Z 81.189,A -85,B 0,C 180,E1 -16868.208,E2 -16868.208} C_VEL
LIN {X 0,Y 291.29,Z 81.202,A -85,B 0,C 180,E1 -16872.498,E2 -16872.498} C_VEL
LIN {X 0,Y 291.292,Z 81.196,A -85,B 0,C 180,E1 -16876.371,E2 -16876.371} C_VEL
LIN {X 0,Y 291.302,Z 81.197,A -85,B 0,C 180,E1 -16879.373,E2 -16879.373} C_VEL
LIN {X 0,Y 290.655,Z 81.279,A -85,B 0,C 180,E1 -16880.527,E2 -16880.527} C_VEL
LIN {X 0,Y 287.858,Z 81.627,A -85,B 0,C 180,E1 -16882.409,E2 -16882.409} C_VEL
LIN {X 0,Y 285.46,Z 81.926,A -85,B 0,C 180,E1 -16883.936,E2 -16883.936} C_VEL
LIN {X 0,Y 284.401,Z 82.054,A -85,B 0,C 180,E1 -16885.117,E2 -16885.117} C_VEL
LIN {X 0,Y 284.298,Z 82.065,A -85,B 0,C 180,E1 -16885.518,E2 -16885.518} C_VEL
LIN {X 0,Y 284.281,Z 82.065,A -85,B 0,C 180,E1 -16888.723,E2 -16888.723} C_VEL
LIN {X 0,Y 284.33,Z 82.058,A -85,B 0,C 180,E1 -16892.854,E2 -16892.854} C_VEL
LIN {X 0,Y 284.331,Z 82.058,A -85,B 0,C 180,E1 -16896.703,E2 -16896.703} C_VEL
LIN {X 0,Y 284.38,Z 82.061,A -85,B 0,C 180,E1 -16899.904,E2 -16899.904} C_VEL
LIN {X 0,Y 284.451,Z 82.051,A -85,B 0,C 180,E1 -16904.492,E2 -16904.492} C_VEL
LIN {X 0,Y 284.47,Z 82.037,A -85,B 0,C 180,E1 -16908.6,E2 -16908.6} C_VEL
LIN {X 0,Y 284.611,Z 82.031,A -85,B 0,C 180,E1 -16911.479,E2 -16911.479} C_VEL
LIN {X 0,Y 284.572,Z 82.023,A -85,B 0,C 180,E1 -16914.33,E2 -16914.33} C_VEL
LIN {X 0,Y 284.842,Z 81.994,A -85,B 0,C 180,E1 -16918.586,E2 -16918.586} C_VEL
LIN {X 0,Y 284.848,Z 81.996,A -85,B 0,C 180,E1 -16921.413,E2 -16921.413} C_VEL
LIN {X 0,Y 284.645,Z 82.019,A -85,B 0,C 180,E1 -16927.091,E2 -16927.091} C_VEL
LIN {X 0,Y 284.517,Z 82.039,A -85,B 0,C 180,E1 -16929.957,E2 -16929.957} C_VEL
LIN {X 0,Y 284.466,Z 82.049,A -85,B 0,C 180,E1 -16934.303,E2 -16934.303} C_VEL
LIN {X 0,Y 284.389,Z 82.055,A -85,B 0,C 180,E1 -16938.739,E2 -16938.739} C_VEL
LIN {X 0,Y 284.369,Z 82.055,A -85,B 0,C 180,E1 -16943.293,E2 -16943.293} C_VEL
LIN {X 0,Y 284.399,Z 82.05,A -85,B 0,C 180,E1 -16947.173,E2 -16947.173} C_VEL
LIN {X 0,Y 284.296,Z 82.064,A -85,B 0,C 180,E1 -16951.274,E2 -16951.274} C_VEL
LIN {X 0,Y 284.343,Z 82.043,A -85,B 0,C 180,E1 -16955.348,E2 -16955.348} C_VEL
LIN {X 0,Y 284.321,Z 82.055,A -85,B 0,C 180,E1 -16958.168,E2 -16958.168} C_VEL
LIN {X 0,Y 284.271,Z 82.075,A -85,B 0,C 180,E1 -16962.124,E2 -16962.124} C_VEL
LIN {X 0,Y 284.257,Z 82.071,A -85,B 0,C 180,E1 -16966.189,E2 -16966.189} C_VEL
LIN {X 0,Y 284.308,Z 82.065,A -85,B 0,C 180,E1 -16970.024,E2 -16970.024} C_VEL
LIN {X 0,Y 284.349,Z 82.188,A -85,B 0,C 180,E1 -16971.328,E2 -16971.328} C_VEL
LIN {X 0,Y 286.761,Z 91.441,A -85,B 0,C 180,E1 -16974.844,E2 -16974.844} C_VEL
LIN {X 0,Y 288.813,Z 100.242,A -85,B 0,C 180,E1 -16977.967,E2 -16977.967} C_VEL
LIN {X 0,Y 289.926,Z 105.116,A -85,B 0,C 180,E1 -16979.577,E2 -16979.577} C_VEL
LIN {X 0,Y 295.596,Z 118.343,A -85,B 0,C 180,E1 -16980.662,E2 -16980.662} C_VEL
LIN {X 0,Y 300.589,Z 145.01,A -85,B 0,C 180,E1 -16981.984,E2 -16981.984} C_VEL
LIN {X 0,Y 302.146,Z 155.904,A -85,B 0,C 180,E1 -16982.453,E2 -16982.453} C_VEL
LIN {X 0,Y 300.268,Z 213.525,A -85,B 0,C 180,E1 -16983.828,E2 -16983.828} C_VEL
LIN {X 0,Y 299.244,Z 226.903,A -85,B 0,C 180,E1 -16984.387,E2 -16984.387} C_VEL
LIN {X 0,Y 297.607,Z 240.243,A -85,B 0,C 180,E1 -16985.218,E2 -16985.218} C_VEL
LIN {X 0,Y 295.894,Z 251.445,A -85,B 0,C 180,E1 -16986.185,E2 -16986.185} C_VEL
LIN {X 0,Y 294.051,Z 261.764,A -85,B 0,C 180,E1 -16987.331,E2 -16987.331} C_VEL
LIN {X 0,Y 291.831,Z 272.444,A -85,B 0,C 180,E1 -16988.823,E2 -16988.823} C_VEL
LIN {X 0,Y 289.692,Z 282.076,A -85,B 0,C 180,E1 -16990.513,E2 -16990.513} C_VEL
LIN {X 0,Y 287.829,Z 290.72,A -85,B 0,C 180,E1 -16992.414,E2 -16992.414} C_VEL
LIN {X 0,Y 286.177,Z 297.757,A -85,B 0,C 180,E1 -16994.327,E2 -16994.327} C_VEL
LIN {X 0,Y 284.67,Z 304.002,A -85,B 0,C 180,E1 -16996.435,E2 -16996.435} C_VEL
LIN {X 0,Y 283.59,Z 308.99,A -85,B 0,C 180,E1 -16998.564,E2 -16998.564} C_VEL
LIN {X 0,Y 282.895,Z 312.865,A -85,B 0,C 180,E1 -17000.707,E2 -17000.707} C_VEL
LIN {X 0,Y 282.499,Z 315.731,A -85,B 0,C 180,E1 -17002.854,E2 -17002.854} C_VEL
LIN {X 0,Y 282.367,Z 318.075,A -85,B 0,C 180,E1 -17005.717,E2 -17005.717} C_VEL
LIN {X 0,Y 282.427,Z 318.665,A -85,B 0,C 180,E1 -17007.147,E2 -17007.147} C_VEL
LIN {X 0,Y 282.43,Z 318.822,A -85,B 0,C 180,E1 -17008.574,E2 -17008.574} C_VEL
LIN {X 0,Y 282.495,Z 318.576,A -85,B 0,C 180,E1 -17010,E2 -17010} C_VEL
LIN {X 0,Y 282.448,Z 317.935,A -85,B 0,C 180,E1 -17011.425,E2 -17011.425} C_VEL
LIN {X 0,Y 282.461,Z 316.901,A -85,B 0,C 180,E1 -17012.852,E2 -17012.852} C_VEL
LIN {X 0,Y 282.384,Z 313.92,A -85,B 0,C 180,E1 -17015.422,E2 -17015.422} C_VEL
LIN {X 0,Y 282.594,Z 309.738,A -85,B 0,C 180,E1 -17017.861,E2 -17017.861} C_VEL
LIN {X 0,Y 282.982,Z 304.855,A -85,B 0,C 180,E1 -17020.011,E2 -17020.011} C_VEL
LIN {X 0,Y 283.634,Z 298.687,A -85,B 0,C 180,E1 -17022.158,E2 -17022.158} C_VEL
LIN {X 0,Y 284.693,Z 291.021,A -85,B 0,C 180,E1 -17024.291,E2 -17024.291} C_VEL
LIN {X 0,Y 285.948,Z 282.516,A -85,B 0,C 180,E1 -17026.186,E2 -17026.186} C_VEL
LIN {X 0,Y 287.084,Z 272.458,A -85,B 0,C 180,E1 -17028.003,E2 -17028.003} C_VEL
LIN {X 0,Y 288.741,Z 261.596,A -85,B 0,C 180,E1 -17029.553,E2 -17029.553} C_VEL
LIN {X 0,Y 290.088,Z 250.985,A -85,B 0,C 180,E1 -17030.751,E2 -17030.751} C_VEL
LIN {X 0,Y 291.471,Z 238.189,A -85,B 0,C 180,E1 -17031.853,E2 -17031.853} C_VEL
LIN {X 0,Y 292.654,Z 225.386,A -85,B 0,C 180,E1 -17032.642,E2 -17032.642} C_VEL
LIN {X 0,Y 293.294,Z 212.944,A -85,B 0,C 180,E1 -17033.149,E2 -17033.149} C_VEL
LIN {X 0,Y 294.619,Z 151.32,A -85,B 0,C 180,E1 -17034.652,E2 -17034.652} C_VEL
LIN {X 0,Y 290.224,Z 117.589,A -85,B 0,C 180,E1 -17035.878,E2 -17035.878} C_VEL
LIN {X 0,Y 288.443,Z 105.654,A -85,B 0,C 180,E1 -17036.362,E2 -17036.362} C_VEL
LIN {X 0,Y 288.591,Z 102.813,A -85,B 0,C 180,E1 -17037.168,E2 -17037.168} C_VEL
LIN {X 0,Y 286.762,Z 93.098,A -85,B 0,C 180,E1 -17040.156,E2 -17040.156} C_VEL
LIN {X 0,Y 284.389,Z 82.066,A -85,B 0,C 180,E1 -17043.781,E2 -17043.781} C_VEL
LIN {X 0,Y 284.335,Z 82.072,A -85,B 0,C 180,E1 -17047.725,E2 -17047.725} C_VEL
LIN {X 0,Y 284.271,Z 82.076,A -85,B 0,C 180,E1 -17051.875,E2 -17051.875} C_VEL
LIN {X 0,Y 284.254,Z 82.076,A -85,B 0,C 180,E1 -17056.189,E2 -17056.189} C_VEL
LIN {X 0,Y 284.305,Z 82.063,A -85,B 0,C 180,E1 -17060.024,E2 -17060.024} C_VEL
LIN {X 0,Y 284.331,Z 82.066,A -85,B 0,C 180,E1 -17063.614,E2 -17063.614} C_VEL
LIN {X 0,Y 284.307,Z 82.072,A -85,B 0,C 180,E1 -17067.189,E2 -17067.189} C_VEL
LIN {X 0,Y 284.358,Z 82.063,A -85,B 0,C 180,E1 -17070.376,E2 -17070.376} C_VEL
LIN {X 0,Y 284.377,Z 82.057,A -85,B 0,C 180,E1 -17073.587,E2 -17073.587} C_VEL
LIN {X 0,Y 284.366,Z 82.065,A -85,B 0,C 180,E1 -17076.707,E2 -17076.707} C_VEL
LIN {X 0,Y 284.403,Z 82.055,A -85,B 0,C 180,E1 -17081.262,E2 -17081.262} C_VEL
LIN {X 0,Y 284.491,Z 82.049,A -85,B 0,C 180,E1 -17084.459,E2 -17084.459} C_VEL
LIN {X 0,Y 284.487,Z 82.044,A -85,B 0,C 180,E1 -17088.602,E2 -17088.602} C_VEL
LIN {X 0,Y 284.638,Z 82.027,A -85,B 0,C 180,E1 -17091.481,E2 -17091.481} C_VEL
LIN {X 0,Y 284.594,Z 82.032,A -85,B 0,C 180,E1 -17094.331,E2 -17094.331} C_VEL
LIN {X 0,Y 284.852,Z 82.001,A -85,B 0,C 180,E1 -17098.587,E2 -17098.587} C_VEL
LIN {X 0,Y 284.852,Z 82,A -85,B 0,C 180,E1 -17101.414,E2 -17101.414} C_VEL
LIN {X 0,Y 284.654,Z 82.022,A -85,B 0,C 180,E1 -17107.092,E2 -17107.092} C_VEL
LIN {X 0,Y 284.513,Z 82.043,A -85,B 0,C 180,E1 -17109.958,E2 -17109.958} C_VEL
LIN {X 0,Y 284.481,Z 82.043,A -85,B 0,C 180,E1 -17114.303,E2 -17114.303} C_VEL
LIN {X 0,Y 284.425,Z 82.055,A -85,B 0,C 180,E1 -17117.249,E2 -17117.249} C_VEL
LIN {X 0,Y 284.379,Z 82.054,A -85,B 0,C 180,E1 -17120.243,E2 -17120.243} C_VEL
LIN {X 0,Y 284.369,Z 82.06,A -85,B 0,C 180,E1 -17123.876,E2 -17123.876} C_VEL
LIN {X 0,Y 284.394,Z 82.06,A -85,B 0,C 180,E1 -17127.173,E2 -17127.173} C_VEL
LIN {X 0,Y 284.294,Z 82.073,A -85,B 0,C 180,E1 -17131.275,E2 -17131.275} C_VEL
LIN {X 0,Y 284.341,Z 82.066,A -85,B 0,C 180,E1 -17135.348,E2 -17135.348} C_VEL
LIN {X 0,Y 284.301,Z 82.069,A -85,B 0,C 180,E1 -17138.171,E2 -17138.171} C_VEL
LIN {X 0,Y 284.238,Z 82.077,A -85,B 0,C 180,E1 -17142.118,E2 -17142.118} C_VEL
LIN {X 0,Y 284.256,Z 82.077,A -85,B 0,C 180,E1 -17146.19,E2 -17146.19} C_VEL
LIN {X 0,Y 284.307,Z 82.07,A -85,B 0,C 180,E1 -17150.025,E2 -17150.025} C_VEL
LIN {X 0,Y 284.323,Z 82.067,A -85,B 0,C 180,E1 -17153.613,E2 -17153.613} C_VEL
LIN {X 0,Y 284.308,Z 82.066,A -85,B 0,C 180,E1 -17157.191,E2 -17157.191} C_VEL
LIN {X 0,Y 284.339,Z 82.06,A -85,B 0,C 180,E1 -17160.374,E2 -17160.374} C_VEL
LIN {X 0,Y 284.302,Z 82.071,A -85,B 0,C 180,E1 -17163.579,E2 -17163.579} C_VEL
LIN {X 0,Y 284.324,Z 82.069,A -85,B 0,C 180,E1 -17166.704,E2 -17166.704} C_VEL
LIN {X 0,Y 284.459,Z 82.228,A -85,B 0,C 180,E1 -17170.178,E2 -17170.178} C_VEL
LIN {X 0,Y 284.632,Z 83.016,A -85,B 0,C 180,E1 -17170.415,E2 -17170.415} C_VEL
LIN {X 0,Y 291.878,Z 101.46,A -85,B 0,C 180,E1 -17171.532,E2 -17171.532} C_VEL
LIN {X 0,Y 295.533,Z 112.062,A -85,B 0,C 180,E1 -17172.106,E2 -17172.106} C_VEL
LIN {X 0,Y 293.671,Z 189.353,A -85,B 0,C 180,E1 -17173.981,E2 -17173.981} C_VEL
LIN {X 0,Y 293.05,Z 202.613,A -85,B 0,C 180,E1 -17174.571,E2 -17174.571} C_VEL
LIN {X 0,Y 292.125,Z 215.856,A -85,B 0,C 180,E1 -17175.457,E2 -17175.457} C_VEL
LIN {X 0,Y 291.073,Z 227.764,A -85,B 0,C 180,E1 -17176.562,E2 -17176.562} C_VEL
LIN {X 0,Y 289.724,Z 239.159,A -85,B 0,C 180,E1 -17177.924,E2 -17177.924} C_VEL
LIN {X 0,Y 288.346,Z 249.432,A -85,B 0,C 180,E1 -17179.467,E2 -17179.467} C_VEL
LIN {X 0,Y 286.932,Z 258.679,A -85,B 0,C 180,E1 -17181.195,E2 -17181.195} C_VEL
LIN {X 0,Y 285.614,Z 267.619,A -85,B 0,C 180,E1 -17183.288,E2 -17183.288} C_VEL
LIN {X 0,Y 284.501,Z 274.833,A -85,B 0,C 180,E1 -17185.396,E2 -17185.396} C_VEL
LIN {X 0,Y 283.861,Z 279.708,A -85,B 0,C 180,E1 -17187.162,E2 -17187.162} C_VEL
LIN {X 0,Y 283.226,Z 284.456,A -85,B 0,C 180,E1 -17189.29,E2 -17189.29} C_VEL
LIN {X 0,Y 282.828,Z 288.103,A -85,B 0,C 180,E1 -17191.424,E2 -17191.424} C_VEL
LIN {X 0,Y 282.63,Z 289.994,A -85,B 0,C 180,E1 -17192.851,E2 -17192.851} C_VEL
LIN {X 0,Y 282.599,Z 291.433,A -85,B 0,C 180,E1 -17194.279,E2 -17194.279} C_VEL
LIN {X 0,Y 282.605,Z 292.546,A -85,B 0,C 180,E1 -17195.87,E2 -17195.87} C_VEL
LIN {X 0,Y 282.496,Z 293.368,A -85,B 0,C 180,E1 -17198.585,E2 -17198.585} C_VEL
LIN {X 0,Y 282.563,Z 293.21,A -85,B 0,C 180,E1 -17200.027,E2 -17200.027} C_VEL
LIN {X 0,Y 283.092,Z 291.684,A -85,B 0,C 180,E1 -17202.911,E2 -17202.911} C_VEL
LIN {X 0,Y 283.695,Z 289.613,A -85,B 0,C 180,E1 -17204.948,E2 -17204.948} C_VEL
LIN {X 0,Y 284.567,Z 286.235,A -85,B 0,C 180,E1 -17207.24,E2 -17207.24} C_VEL
LIN {X 0,Y 285.703,Z 281.921,A -85,B 0,C 180,E1 -17209.396,E2 -17209.396} C_VEL
LIN {X 0,Y 287.121,Z 276.385,A -85,B 0,C 180,E1 -17211.541,E2 -17211.541} C_VEL
LIN {X 0,Y 288.905,Z 269.436,A -85,B 0,C 180,E1 -17213.665,E2 -17213.665} C_VEL
LIN {X 0,Y 290.976,Z 260.667,A -85,B 0,C 180,E1 -17215.77,E2 -17215.77} C_VEL
LIN {X 0,Y 293.119,Z 250.66,A -85,B 0,C 180,E1 -17217.681,E2 -17217.681} C_VEL
LIN {X 0,Y 295.068,Z 240.392,A -85,B 0,C 180,E1 -17219.228,E2 -17219.228} C_VEL
LIN {X 0,Y 297.028,Z 228.944,A -85,B 0,C 180,E1 -17220.579,E2 -17220.579} C_VEL
LIN {X 0,Y 298.698,Z 217.233,A -85,B 0,C 180,E1 -17221.646,E2 -17221.646} C_VEL
LIN {X 0,Y 299.942,Z 204.569,A -85,B 0,C 180,E1 -17222.504,E2 -17222.504} C_VEL
LIN {X 0,Y 300.984,Z 191.049,A -85,B 0,C 180,E1 -17223.102,E2 -17223.102} C_VEL
LIN {X 0,Y 302.323,Z 148.321,A -85,B 0,C 180,E1 -17224.156,E2 -17224.156} C_VEL
LIN {X 0,Y 303.081,Z 121.872,A -85,B 0,C 180,E1 -17224.787,E2 -17224.787} C_VEL
LIN {X 0,Y 295.009,Z 103.623,A -85,B 0,C 180,E1 -17226.248,E2 -17226.248} C_VEL
LIN {X 0,Y 286.498,Z 87.197,A -85,B 0,C 180,E1 -17227.825,E2 -17227.825} C_VEL
LIN {X 0,Y 284.724,Z 83.725,A -85,B 0,C 180,E1 -17228.182,E2 -17228.182} C_VEL
LIN {X 0,Y 284.308,Z 82.073,A -85,B 0,C 180,E1 -17228.954,E2 -17228.954} C_VEL
LIN {X 0,Y 284.24,Z 82.079,A -85,B 0,C 180,E1 -17232.117,E2 -17232.117} C_VEL
LIN {X 0,Y 284.241,Z 82.071,A -85,B 0,C 180,E1 -17236.186,E2 -17236.186} C_VEL
LIN {X 0,Y 284.286,Z 82.074,A -85,B 0,C 180,E1 -17240.03,E2 -17240.03} C_VEL
LIN {X 0,Y 284.321,Z 82.067,A -85,B 0,C 180,E1 -17243.612,E2 -17243.612} C_VEL
LIN {X 0,Y 284.298,Z 82.065,A -85,B 0,C 180,E1 -17245.518,E2 -17245.518} C_VEL
LIN {X 0,Y 283.583,Z 82.161,A -85,B 0,C 180,E1 -17246.701,E2 -17246.701} C_VEL
LIN {X 0,Y 280.702,Z 82.515,A -85,B 0,C 180,E1 -17248.627,E2 -17248.627} C_VEL
LIN {X 0,Y 278.302,Z 82.818,A -85,B 0,C 180,E1 -17250.192,E2 -17250.192} C_VEL
LIN {X 0,Y 277.298,Z 82.939,A -85,B 0,C 180,E1 -17251.405,E2 -17251.405} C_VEL
LIN {X 0,Y 277.228,Z 82.944,A -85,B 0,C 180,E1 -17251.815,E2 -17251.815} C_VEL
LIN {X 0,Y 277.285,Z 82.942,A -85,B 0,C 180,E1 -17256.075,E2 -17256.075} C_VEL
LIN {X 0,Y 277.332,Z 82.936,A -85,B 0,C 180,E1 -17260.765,E2 -17260.765} C_VEL
LIN {X 0,Y 277.413,Z 82.929,A -85,B 0,C 180,E1 -17265.324,E2 -17265.324} C_VEL
LIN {X 0,Y 277.458,Z 82.92,A -85,B 0,C 180,E1 -17269.787,E2 -17269.787} C_VEL
LIN {X 0,Y 277.602,Z 82.895,A -85,B 0,C 180,E1 -17272.727,E2 -17272.727} C_VEL
LIN {X 0,Y 277.809,Z 82.87,A -85,B 0,C 180,E1 -17278.55,E2 -17278.55} C_VEL
LIN {X 0,Y 277.814,Z 82.873,A -85,B 0,C 180,E1 -17281.449,E2 -17281.449} C_VEL
LIN {X 0,Y 277.604,Z 82.896,A -85,B 0,C 180,E1 -17287.272,E2 -17287.272} C_VEL
LIN {X 0,Y 277.46,Z 82.916,A -85,B 0,C 180,E1 -17290.213,E2 -17290.213} C_VEL
LIN {X 0,Y 277.412,Z 82.927,A -85,B 0,C 180,E1 -17294.675,E2 -17294.675} C_VEL
LIN {X 0,Y 277.338,Z 82.936,A -85,B 0,C 180,E1 -17299.234,E2 -17299.234} C_VEL
LIN {X 0,Y 277.322,Z 82.94,A -85,B 0,C 180,E1 -17304.17,E2 -17304.17} C_VEL
LIN {X 0,Y 277.327,Z 82.932,A -85,B 0,C 180,E1 -17307.504,E2 -17307.504} C_VEL
LIN {X 0,Y 277.274,Z 82.94,A -85,B 0,C 180,E1 -17310.481,E2 -17310.481} C_VEL
LIN {X 0,Y 277.249,Z 82.947,A -85,B 0,C 180,E1 -17313.895,E2 -17313.895} C_VEL
LIN {X 0,Y 277.274,Z 82.921,A -85,B 0,C 180,E1 -17317.468,E2 -17317.468} C_VEL
LIN {X 0,Y 277.212,Z 82.95,A -85,B 0,C 180,E1 -17321.236,E2 -17321.236} C_VEL
LIN {X 0,Y 277.202,Z 82.954,A -85,B 0,C 180,E1 -17325.226,E2 -17325.226} C_VEL
LIN {X 0,Y 277.225,Z 82.95,A -85,B 0,C 180,E1 -17329.512,E2 -17329.512} C_VEL
LIN {X 0,Y 277.291,Z 83.012,A -85,B 0,C 180,E1 -17330.463,E2 -17330.463} C_VEL
LIN {X 0,Y 279.881,Z 92.88,A -85,B 0,C 180,E1 -17334.352,E2 -17334.352} C_VEL
LIN {X 0,Y 282.121,Z 102.554,A -85,B 0,C 180,E1 -17337.885,E2 -17337.885} C_VEL
LIN {X 0,Y 282.63,Z 104.818,A -85,B 0,C 180,E1 -17338.599,E2 -17338.599} C_VEL
LIN {X 0,Y 289.707,Z 120.46,A -85,B 0,C 180,E1 -17339.993,E2 -17339.993} C_VEL
LIN {X 0,Y 294.182,Z 144.371,A -85,B 0,C 180,E1 -17341.224,E2 -17341.224} C_VEL
LIN {X 0,Y 296.013,Z 157.225,A -85,B 0,C 180,E1 -17341.797,E2 -17341.797} C_VEL
LIN {X 0,Y 294.037,Z 213.947,A -85,B 0,C 180,E1 -17343.182,E2 -17343.182} C_VEL
LIN {X 0,Y 292.898,Z 227.82,A -85,B 0,C 180,E1 -17343.79,E2 -17343.79} C_VEL
LIN {X 0,Y 291.196,Z 240.788,A -85,B 0,C 180,E1 -17344.634,E2 -17344.634} C_VEL
LIN {X 0,Y 289.107,Z 253.347,A -85,B 0,C 180,E1 -17345.781,E2 -17345.781} C_VEL
LIN {X 0,Y 287.004,Z 264.547,A -85,B 0,C 180,E1 -17347.123,E2 -17347.123} C_VEL
LIN {X 0,Y 284.75,Z 274.657,A -85,B 0,C 180,E1 -17348.65,E2 -17348.65} C_VEL
LIN {X 0,Y 282.582,Z 283.786,A -85,B 0,C 180,E1 -17350.381,E2 -17350.381} C_VEL
LIN {X 0,Y 280.55,Z 292.704,A -85,B 0,C 180,E1 -17352.505,E2 -17352.505} C_VEL
LIN {X 0,Y 278.833,Z 299.903,A -85,B 0,C 180,E1 -17354.653,E2 -17354.653} C_VEL
LIN {X 0,Y 277.276,Z 305.669,A -85,B 0,C 180,E1 -17356.813,E2 -17356.813} C_VEL
LIN {X 0,Y 276.322,Z 310.234,A -85,B 0,C 180,E1 -17359.003,E2 -17359.003} C_VEL
LIN {X 0,Y 275.699,Z 313.726,A -85,B 0,C 180,E1 -17361.202,E2 -17361.202} C_VEL
LIN {X 0,Y 275.448,Z 315.483,A -85,B 0,C 180,E1 -17362.67,E2 -17362.67} C_VEL
LIN {X 0,Y 275.274,Z 317.794,A -85,B 0,C 180,E1 -17365.607,E2 -17365.607} C_VEL
LIN {X 0,Y 275.33,Z 318.362,A -85,B 0,C 180,E1 -17367.073,E2 -17367.073} C_VEL
LIN {X 0,Y 275.351,Z 318.494,A -85,B 0,C 180,E1 -17368.537,E2 -17368.537} C_VEL
LIN {X 0,Y 275.41,Z 318.232,A -85,B 0,C 180,E1 -17370,E2 -17370} C_VEL
LIN {X 0,Y 275.368,Z 317.575,A -85,B 0,C 180,E1 -17371.462,E2 -17371.462} C_VEL
LIN {X 0,Y 275.385,Z 316.522,A -85,B 0,C 180,E1 -17372.925,E2 -17372.925} C_VEL
LIN {X 0,Y 275.288,Z 313.814,A -85,B 0,C 180,E1 -17375.342,E2 -17375.342} C_VEL
LIN {X 0,Y 275.521,Z 309.271,A -85,B 0,C 180,E1 -17378.064,E2 -17378.064} C_VEL
LIN {X 0,Y 275.934,Z 304.348,A -85,B 0,C 180,E1 -17380.27,E2 -17380.27} C_VEL
LIN {X 0,Y 276.636,Z 298.136,A -85,B 0,C 180,E1 -17382.47,E2 -17382.47} C_VEL
LIN {X 0,Y 277.743,Z 290.407,A -85,B 0,C 180,E1 -17384.657,E2 -17384.657} C_VEL
LIN {X 0,Y 279.154,Z 281.121,A -85,B 0,C 180,E1 -17386.738,E2 -17386.738} C_VEL
LIN {X 0,Y 280.46,Z 270.615,A -85,B 0,C 180,E1 -17388.632,E2 -17388.632} C_VEL
LIN {X 0,Y 282.267,Z 259.292,A -85,B 0,C 180,E1 -17390.21,E2 -17390.21} C_VEL
LIN {X 0,Y 283.632,Z 248.154,A -85,B 0,C 180,E1 -17391.437,E2 -17391.437} C_VEL
LIN {X 0,Y 284.981,Z 235.797,A -85,B 0,C 180,E1 -17392.473,E2 -17392.473} C_VEL
LIN {X 0,Y 286.146,Z 222.724,A -85,B 0,C 180,E1 -17393.235,E2 -17393.235} C_VEL
LIN {X 0,Y 286.727,Z 210.169,A -85,B 0,C 180,E1 -17393.71,E2 -17393.71} C_VEL
LIN {X 0,Y 288.003,Z 152.109,A -85,B 0,C 180,E1 -17395.149,E2 -17395.149} C_VEL
LIN {X 0,Y 283.735,Z 118.797,A -85,B 0,C 180,E1 -17396.394,E2 -17396.394} C_VEL
LIN {X 0,Y 281.696,Z 105.34,A -85,B 0,C 180,E1 -17396.954,E2 -17396.954} C_VEL
LIN {X 0,Y 280.498,Z 97.593,A -85,B 0,C 180,E1 -17399.362,E2 -17399.362} C_VEL
LIN {X 0,Y 277.818,Z 85.306,A -85,B 0,C 180,E1 -17403.404,E2 -17403.404} C_VEL
LIN {X 0,Y 277.332,Z 82.945,A -85,B 0,C 180,E1 -17404.212,E2 -17404.212} C_VEL
LIN {X 0,Y 277.275,Z 82.948,A -85,B 0,C 180,E1 -17408.21,E2 -17408.21} C_VEL
LIN {X 0,Y 277.214,Z 82.953,A -85,B 0,C 180,E1 -17412.675,E2 -17412.675} C_VEL
LIN {X 0,Y 277.208,Z 82.954,A -85,B 0,C 180,E1 -17416.802,E2 -17416.802} C_VEL
LIN {X 0,Y 277.233,Z 82.942,A -85,B 0,C 180,E1 -17420.672,E2 -17420.672} C_VEL
LIN {X 0,Y 277.283,Z 82.942,A -85,B 0,C 180,E1 -17424.341,E2 -17424.341} C_VEL
LIN {X 0,Y 277.244,Z 82.949,A -85,B 0,C 180,E1 -17427.836,E2 -17427.836} C_VEL
LIN {X 0,Y 277.288,Z 82.944,A -85,B 0,C 180,E1 -17431.213,E2 -17431.213} C_VEL
LIN {X 0,Y 277.313,Z 82.938,A -85,B 0,C 180,E1 -17434.48,E2 -17434.48} C_VEL
LIN {X 0,Y 277.285,Z 82.942,A -85,B 0,C 180,E1 -17437.655,E2 -17437.655} C_VEL
LIN {X 0,Y 277.344,Z 82.933,A -85,B 0,C 180,E1 -17440.766,E2 -17440.766} C_VEL
LIN {X 0,Y 277.434,Z 82.922,A -85,B 0,C 180,E1 -17445.326,E2 -17445.326} C_VEL
LIN {X 0,Y 277.46,Z 82.919,A -85,B 0,C 180,E1 -17449.787,E2 -17449.787} C_VEL
LIN {X 0,Y 277.64,Z 82.9,A -85,B 0,C 180,E1 -17452.729,E2 -17452.729} C_VEL
LIN {X 0,Y 277.818,Z 82.877,A -85,B 0,C 180,E1 -17458.551,E2 -17458.551} C_VEL
LIN {X 0,Y 277.818,Z 82.877,A -85,B 0,C 180,E1 -17461.45,E2 -17461.45} C_VEL
LIN {X 0,Y 277.611,Z 82.9,A -85,B 0,C 180,E1 -17467.272,E2 -17467.272} C_VEL
LIN {X 0,Y 277.457,Z 82.92,A -85,B 0,C 180,E1 -17470.214,E2 -17470.214} C_VEL
LIN {X 0,Y 277.434,Z 82.919,A -85,B 0,C 180,E1 -17474.675,E2 -17474.675} C_VEL
LIN {X 0,Y 277.345,Z 82.936,A -85,B 0,C 180,E1 -17479.234,E2 -17479.234} C_VEL
LIN {X 0,Y 277.319,Z 82.938,A -85,B 0,C 180,E1 -17484.171,E2 -17484.171} C_VEL
LIN {X 0,Y 277.323,Z 82.94,A -85,B 0,C 180,E1 -17487.505,E2 -17487.505} C_VEL
LIN {X 0,Y 277.272,Z 82.945,A -85,B 0,C 180,E1 -17490.482,E2 -17490.482} C_VEL
LIN {X 0,Y 277.247,Z 82.947,A -85,B 0,C 180,E1 -17493.896,E2 -17493.896} C_VEL
LIN {X 0,Y 277.261,Z 82.946,A -85,B 0,C 180,E1 -17497.471,E2 -17497.471} C_VEL
LIN {X 0,Y 277.184,Z 82.957,A -85,B 0,C 180,E1 -17501.242,E2 -17501.242} C_VEL
LIN {X 0,Y 277.199,Z 82.955,A -85,B 0,C 180,E1 -17505.228,E2 -17505.228} C_VEL
LIN {X 0,Y 277.222,Z 82.951,A -85,B 0,C 180,E1 -17509.513,E2 -17509.513} C_VEL
LIN {X 0,Y 277.258,Z 82.95,A -85,B 0,C 180,E1 -17512.53,E2 -17512.53} C_VEL
LIN {X 0,Y 277.247,Z 82.951,A -85,B 0,C 180,E1 -17516.105,E2 -17516.105} C_VEL
LIN {X 0,Y 277.264,Z 82.946,A -85,B 0,C 180,E1 -17519.539,E2 -17519.539} C_VEL
LIN {X 0,Y 277.291,Z 82.943,A -85,B 0,C 180,E1 -17522.857,E2 -17522.857} C_VEL
LIN {X 0,Y 277.275,Z 82.949,A -85,B 0,C 180,E1 -17526.075,E2 -17526.075} C_VEL
LIN {X 0,Y 277.371,Z 83.142,A -85,B 0,C 180,E1 -17529.732,E2 -17529.732} C_VEL
LIN {X 0,Y 278.564,Z 86.097,A -85,B 0,C 180,E1 -17529.943,E2 -17529.943} C_VEL
LIN {X 0,Y 284.464,Z 100.763,A -85,B 0,C 180,E1 -17530.88,E2 -17530.88} C_VEL
LIN {X 0,Y 288.96,Z 113.647,A -85,B 0,C 180,E1 -17531.611,E2 -17531.611} C_VEL
LIN {X 0,Y 287.031,Z 190.063,A -85,B 0,C 180,E1 -17533.509,E2 -17533.509} C_VEL
LIN {X 0,Y 286.361,Z 203.191,A -85,B 0,C 180,E1 -17534.11,E2 -17534.11} C_VEL
LIN {X 0,Y 285.423,Z 216.358,A -85,B 0,C 180,E1 -17535.017,E2 -17535.017} C_VEL
LIN {X 0,Y 284.395,Z 227.433,A -85,B 0,C 180,E1 -17536.058,E2 -17536.058} C_VEL
LIN {X 0,Y 283.009,Z 238.945,A -85,B 0,C 180,E1 -17537.451,E2 -17537.451} C_VEL
LIN {X 0,Y 281.575,Z 249.308,A -85,B 0,C 180,E1 -17539.029,E2 -17539.029} C_VEL
LIN {X 0,Y 280.233,Z 257.794,A -85,B 0,C 180,E1 -17540.619,E2 -17540.619} C_VEL
LIN {X 0,Y 279.015,Z 265.613,A -85,B 0,C 180,E1 -17542.401,E2 -17542.401} C_VEL
LIN {X 0,Y 277.822,Z 273.258,A -85,B 0,C 180,E1 -17544.557,E2 -17544.557} C_VEL
LIN {X 0,Y 276.789,Z 280.291,A -85,B 0,C 180,E1 -17547.09,E2 -17547.09} C_VEL
LIN {X 0,Y 276.153,Z 284.982,A -85,B 0,C 180,E1 -17549.271,E2 -17549.271} C_VEL
LIN {X 0,Y 275.724,Z 288.579,A -85,B 0,C 180,E1 -17551.461,E2 -17551.461} C_VEL
LIN {X 0,Y 275.549,Z 290.44,A -85,B 0,C 180,E1 -17552.924,E2 -17552.924} C_VEL
LIN {X 0,Y 275.516,Z 291.835,A -85,B 0,C 180,E1 -17554.389,E2 -17554.389} C_VEL
LIN {X 0,Y 275.533,Z 292.834,A -85,B 0,C 180,E1 -17555.856,E2 -17555.856} C_VEL
LIN {X 0,Y 275.451,Z 293.458,A -85,B 0,C 180,E1 -17557.33,E2 -17557.33} C_VEL
LIN {X 0,Y 275.404,Z 293.697,A -85,B 0,C 180,E1 -17558.808,E2 -17558.808} C_VEL
LIN {X 0,Y 275.514,Z 293.498,A -85,B 0,C 180,E1 -17560.286,E2 -17560.286} C_VEL
LIN {X 0,Y 276.095,Z 291.925,A -85,B 0,C 180,E1 -17563.244,E2 -17563.244} C_VEL
LIN {X 0,Y 276.66,Z 290.047,A -85,B 0,C 180,E1 -17565.132,E2 -17565.132} C_VEL
LIN {X 0,Y 277.673,Z 286.377,A -85,B 0,C 180,E1 -17567.682,E2 -17567.682} C_VEL
LIN {X 0,Y 278.893,Z 282.007,A -85,B 0,C 180,E1 -17569.889,E2 -17569.889} C_VEL
LIN {X 0,Y 280.424,Z 276.411,A -85,B 0,C 180,E1 -17572.082,E2 -17572.082} C_VEL
LIN {X 0,Y 282.303,Z 269.37,A -85,B 0,C 180,E1 -17574.254,E2 -17574.254} C_VEL
LIN {X 0,Y 284.489,Z 260.508,A -85,B 0,C 180,E1 -17576.403,E2 -17576.403} C_VEL
LIN {X 0,Y 286.533,Z 251.386,A -85,B 0,C 180,E1 -17578.175,E2 -17578.175} C_VEL
LIN {X 0,Y 288.294,Z 242.481,A -85,B 0,C 180,E1 -17579.581,E2 -17579.581} C_VEL
LIN {X 0,Y 290.331,Z 231.53,A -85,B 0,C 180,E1 -17580.958,E2 -17580.958} C_VEL
LIN {X 0,Y 292.152,Z 219.776,A -85,B 0,C 180,E1 -17582.097,E2 -17582.097} C_VEL
LIN {X 0,Y 293.524,Z 207.313,A -85,B 0,C 180,E1 -17583.016,E2 -17583.016} C_VEL
LIN {X 0,Y 294.562,Z 195.136,A -85,B 0,C 180,E1 -17583.632,E2 -17583.632} C_VEL
LIN {X 0,Y 295.203,Z 180.52,A -85,B 0,C 180,E1 -17584.074,E2 -17584.074} C_VEL
LIN {X 0,Y 296.95,Z 123.802,A -85,B 0,C 180,E1 -17585.446,E2 -17585.446} C_VEL
LIN {X 0,Y 289.055,Z 105.962,A -85,B 0,C 180,E1 -17586.935,E2 -17586.935} C_VEL
LIN {X 0,Y 280.916,Z 90.46,A -85,B 0,C 180,E1 -17588.499,E2 -17588.499} C_VEL
LIN {X 0,Y 277.489,Z 84.06,A -85,B 0,C 180,E1 -17589.224,E2 -17589.224} C_VEL
LIN {X 0,Y 277.258,Z 82.948,A -85,B 0,C 180,E1 -17589.758,E2 -17589.758} C_VEL
LIN {X 0,Y 277.194,Z 82.951,A -85,B 0,C 180,E1 -17593.202,E2 -17593.202} C_VEL
LIN {X 0,Y 277.195,Z 82.959,A -85,B 0,C 180,E1 -17597.33,E2 -17597.33} C_VEL
LIN {X 0,Y 277.253,Z 82.945,A -85,B 0,C 180,E1 -17601.796,E2 -17601.796} C_VEL
LIN {X 0,Y 277.23,Z 82.947,A -85,B 0,C 180,E1 -17605.52,E2 -17605.52} C_VEL
LIN {X 0,Y 277.231,Z 82.948,A -85,B 0,C 180,E1 -17609.534,E2 -17609.534} C_VEL
LIN {X 0,Y 277.228,Z 82.944,A -85,B 0,C 180,E1 -17611.815,E2 -17611.815} C_VEL
LIN {X 0,Y 276.582,Z 83.025,A -85,B 0,C 180,E1 -17613.028,E2 -17613.028} C_VEL
LIN {X 0,Y 273.709,Z 83.393,A -85,B 0,C 180,E1 -17615.004,E2 -17615.004} C_VEL
LIN {X 0,Y 271.274,Z 83.687,A -85,B 0,C 180,E1 -17616.609,E2 -17616.609} C_VEL
LIN {X 0,Y 270.257,Z 83.81,A -85,B 0,C 180,E1 -17617.854,E2 -17617.854} C_VEL
LIN {X 0,Y 270.19,Z 83.82,A -85,B 0,C 180,E1 -17618.276,E2 -17618.276} C_VEL
LIN {X 0,Y 270.269,Z 83.807,A -85,B 0,C 180,E1 -17621.817,E2 -17621.817} C_VEL
LIN {X 0,Y 270.381,Z 83.807,A -85,B 0,C 180,E1 -17624.934,E2 -17624.934} C_VEL
LIN {X 0,Y 270.41,Z 83.797,A -85,B 0,C 180,E1 -17629.517,E2 -17629.517} C_VEL
LIN {X 0,Y 270.564,Z 83.773,A -85,B 0,C 180,E1 -17632.537,E2 -17632.537} C_VEL
LIN {X 0,Y 270.774,Z 83.747,A -85,B 0,C 180,E1 -17638.512,E2 -17638.512} C_VEL
LIN {X 0,Y 270.779,Z 83.749,A -85,B 0,C 180,E1 -17641.487,E2 -17641.487} C_VEL
LIN {X 0,Y 270.565,Z 83.774,A -85,B 0,C 180,E1 -17647.462,E2 -17647.462} C_VEL
LIN {X 0,Y 270.413,Z 83.792,A -85,B 0,C 180,E1 -17650.482,E2 -17650.482} C_VEL
LIN {X 0,Y 270.38,Z 83.804,A -85,B 0,C 180,E1 -17655.066,E2 -17655.066} C_VEL
LIN {X 0,Y 270.299,Z 83.816,A -85,B 0,C 180,E1 -17659.755,E2 -17659.755} C_VEL
LIN {X 0,Y 270.277,Z 83.818,A -85,B 0,C 180,E1 -17664.585,E2 -17664.585} C_VEL
LIN {X 0,Y 270.274,Z 83.814,A -85,B 0,C 180,E1 -17667.908,E2 -17667.908} C_VEL
LIN {X 0,Y 270.186,Z 83.822,A -85,B 0,C 180,E1 -17671.348,E2 -17671.348} C_VEL
LIN {X 0,Y 270.204,Z 83.808,A -85,B 0,C 180,E1 -17674.905,E2 -17674.905} C_VEL
LIN {X 0,Y 270.199,Z 83.821,A -85,B 0,C 180,E1 -17678.71,E2 -17678.71} C_VEL
LIN {X 0,Y 270.174,Z 83.833,A -85,B 0,C 180,E1 -17682.558,E2 -17682.558} C_VEL
LIN {X 0,Y 270.167,Z 83.827,A -85,B 0,C 180,E1 -17686.751,E2 -17686.751} C_VEL
LIN {X 0,Y 270.217,Z 83.896,A -85,B 0,C 180,E1 -17689.561,E2 -17689.561} C_VEL
LIN {X 0,Y 272.921,Z 93.916,A -85,B 0,C 180,E1 -17693.681,E2 -17693.681} C_VEL
LIN {X 0,Y 275.276,Z 104.013,A -85,B 0,C 180,E1 -17697.497,E2 -17697.497} C_VEL
LIN {X 0,Y 279.229,Z 112.534,A -85,B 0,C 180,E1 -17698.362,E2 -17698.362} C_VEL
LIN {X 0,Y 284.113,Z 123.537,A -85,B 0,C 180,E1 -17699.358,E2 -17699.358} C_VEL
LIN {X 0,Y 288.688,Z 149.006,A -85,B 0,C 180,E1 -17700.689,E2 -17700.689} C_VEL
LIN {X 0,Y 289.87,Z 157.086,A -85,B 0,C 180,E1 -17701.066,E2 -17701.066} C_VEL
LIN {X 0,Y 287.921,Z 213.243,A -85,B 0,C 180,E1 -17702.467,E2 -17702.467} C_VEL
LIN {X 0,Y 286.845,Z 226.479,A -85,B 0,C 180,E1 -17703.046,E2 -17703.046} C_VEL
LIN {X 0,Y 285.165,Z 239.198,A -85,B 0,C 180,E1 -17703.861,E2 -17703.861} C_VEL
LIN {X 0,Y 283.334,Z 250.509,A -85,B 0,C 180,E1 -17704.863,E2 -17704.863} C_VEL
LIN {X 0,Y 281.023,Z 262.177,A -85,B 0,C 180,E1 -17706.217,E2 -17706.217} C_VEL
LIN {X 0,Y 278.656,Z 272.673,A -85,B 0,C 180,E1 -17707.77,E2 -17707.77} C_VEL
LIN {X 0,Y 276.338,Z 282.154,A -85,B 0,C 180,E1 -17709.531,E2 -17709.531} C_VEL
LIN {X 0,Y 274.292,Z 290.386,A -85,B 0,C 180,E1 -17711.446,E2 -17711.446} C_VEL
LIN {X 0,Y 272.452,Z 297.567,A -85,B 0,C 180,E1 -17713.515,E2 -17713.515} C_VEL
LIN {X 0,Y 270.845,Z 303.726,A -85,B 0,C 180,E1 -17715.728,E2 -17715.728} C_VEL
LIN {X 0,Y 269.584,Z 308.634,A -85,B 0,C 180,E1 -17717.962,E2 -17717.962} C_VEL
LIN {X 0,Y 268.828,Z 312.437,A -85,B 0,C 180,E1 -17720.216,E2 -17720.216} C_VEL
LIN {X 0,Y 268.37,Z 315.234,A -85,B 0,C 180,E1 -17722.476,E2 -17722.476} C_VEL
LIN {X 0,Y 268.186,Z 317.513,A -85,B 0,C 180,E1 -17725.49,E2 -17725.49} C_VEL
LIN {X 0,Y 268.236,Z 318.055,A -85,B 0,C 180,E1 -17726.996,E2 -17726.996} C_VEL
LIN {X 0,Y 268.272,Z 318.166,A -85,B 0,C 180,E1 -17728.498,E2 -17728.498} C_VEL
LIN {X 0,Y 268.328,Z 317.887,A -85,B 0,C 180,E1 -17730,E2 -17730} C_VEL
LIN {X 0,Y 268.29,Z 317.214,A -85,B 0,C 180,E1 -17731.501,E2 -17731.501} C_VEL
LIN {X 0,Y 268.288,Z 316.136,A -85,B 0,C 180,E1 -17733.003,E2 -17733.003} C_VEL
LIN {X 0,Y 268.21,Z 313.638,A -85,B 0,C 180,E1 -17735.299,E2 -17735.299} C_VEL
LIN {X 0,Y 268.357,Z 310.219,A -85,B 0,C 180,E1 -17737.524,E2 -17737.524} C_VEL
LIN {X 0,Y 268.719,Z 305.653,A -85,B 0,C 180,E1 -17739.787,E2 -17739.787} C_VEL
LIN {X 0,Y 269.525,Z 298.716,A -85,B 0,C 180,E1 -17742.422,E2 -17742.422} C_VEL
LIN {X 0,Y 270.639,Z 291.192,A -85,B 0,C 180,E1 -17744.666,E2 -17744.666} C_VEL
LIN {X 0,Y 272.03,Z 282.479,A -85,B 0,C 180,E1 -17746.75,E2 -17746.75} C_VEL
LIN {X 0,Y 273.187,Z 273.094,A -85,B 0,C 180,E1 -17748.563,E2 -17748.563} C_VEL
LIN {X 0,Y 274.923,Z 262.496,A -85,B 0,C 180,E1 -17750.188,E2 -17750.188} C_VEL
LIN {X 0,Y 276.54,Z 250.658,A -85,B 0,C 180,E1 -17751.623,E2 -17751.623} C_VEL
LIN {X 0,Y 278.047,Z 237.965,A -85,B 0,C 180,E1 -17752.77,E2 -17752.77} C_VEL
LIN {X 0,Y 279.334,Z 224.524,A -85,B 0,C 180,E1 -17753.639,E2 -17753.639} C_VEL
LIN {X 0,Y 280.059,Z 211.589,A -85,B 0,C 180,E1 -17754.174,E2 -17754.174} C_VEL
LIN {X 0,Y 281.438,Z 152.901,A -85,B 0,C 180,E1 -17755.667,E2 -17755.667} C_VEL
LIN {X 0,Y 277.325,Z 120.445,A -85,B 0,C 180,E1 -17756.915,E2 -17756.915} C_VEL
LIN {X 0,Y 275.1,Z 106.801,A -85,B 0,C 180,E1 -17757.501,E2 -17757.501} C_VEL
LIN {X 0,Y 274.604,Z 104.919,A -85,B 0,C 180,E1 -17757.637,E2 -17757.637} C_VEL
LIN {X 0,Y 272.9,Z 95.893,A -85,B 0,C 180,E1 -17760.571,E2 -17760.571} C_VEL
LIN {X 0,Y 270.259,Z 83.826,A -85,B 0,C 180,E1 -17764.744,E2 -17764.744} C_VEL
LIN {X 0,Y 270.221,Z 83.825,A -85,B 0,C 180,E1 -17768.717,E2 -17768.717} C_VEL
LIN {X 0,Y 270.164,Z 83.833,A -85,B 0,C 180,E1 -17773.249,E2 -17773.249} C_VEL
LIN {X 0,Y 270.17,Z 83.833,A -85,B 0,C 180,E1 -17777.442,E2 -17777.442} C_VEL
LIN {X 0,Y 270.206,Z 83.814,A -85,B 0,C 180,E1 -17781.374,E2 -17781.374} C_VEL
LIN {X 0,Y 270.201,Z 83.828,A -85,B 0,C 180,E1 -17785.095,E2 -17785.095} C_VEL
LIN {X 0,Y 270.199,Z 83.829,A -85,B 0,C 180,E1 -17789.13,E2 -17789.13} C_VEL
LIN {X 0,Y 270.264,Z 83.816,A -85,B 0,C 180,E1 -17792.146,E2 -17792.146} C_VEL
LIN {X 0,Y 270.276,Z 83.817,A -85,B 0,C 180,E1 -17795.519,E2 -17795.519} C_VEL
LIN {X 0,Y 270.301,Z 83.807,A -85,B 0,C 180,E1 -17800.245,E2 -17800.245} C_VEL
LIN {X 0,Y 270.402,Z 83.8,A -85,B 0,C 180,E1 -17804.936,E2 -17804.936} C_VEL
LIN {X 0,Y 270.412,Z 83.796,A -85,B 0,C 180,E1 -17809.518,E2 -17809.518} C_VEL
LIN {X 0,Y 270.598,Z 83.778,A -85,B 0,C 180,E1 -17812.539,E2 -17812.539} C_VEL
LIN {X 0,Y 270.784,Z 83.753,A -85,B 0,C 180,E1 -17818.513,E2 -17818.513} C_VEL
LIN {X 0,Y 270.784,Z 83.753,A -85,B 0,C 180,E1 -17821.488,E2 -17821.488} C_VEL
LIN {X 0,Y 270.571,Z 83.778,A -85,B 0,C 180,E1 -17827.463,E2 -17827.463} C_VEL
LIN {X 0,Y 270.409,Z 83.797,A -85,B 0,C 180,E1 -17830.483,E2 -17830.483} C_VEL
LIN {X 0,Y 270.403,Z 83.796,A -85,B 0,C 180,E1 -17835.065,E2 -17835.065} C_VEL
LIN {X 0,Y 270.302,Z 83.809,A -85,B 0,C 180,E1 -17839.756,E2 -17839.756} C_VEL
LIN {X 0,Y 270.274,Z 83.815,A -85,B 0,C 180,E1 -17844.586,E2 -17844.586} C_VEL
LIN {X 0,Y 270.27,Z 83.817,A -85,B 0,C 180,E1 -17847.909,E2 -17847.909} C_VEL
LIN {X 0,Y 270.184,Z 83.83,A -85,B 0,C 180,E1 -17851.349,E2 -17851.349} C_VEL
LIN {X 0,Y 270.201,Z 83.828,A -85,B 0,C 180,E1 -17854.906,E2 -17854.906} C_VEL
LIN {X 0,Y 270.198,Z 83.828,A -85,B 0,C 180,E1 -17858.711,E2 -17858.711} C_VEL
LIN {X 0,Y 270.149,Z 83.834,A -85,B 0,C 180,E1 -17863.246,E2 -17863.246} C_VEL
LIN {X 0,Y 270.171,Z 83.828,A -85,B 0,C 180,E1 -17867.442,E2 -17867.442} C_VEL
LIN {X 0,Y 270.208,Z 83.825,A -85,B 0,C 180,E1 -17871.375,E2 -17871.375} C_VEL
LIN {X 0,Y 270.2,Z 83.826,A -85,B 0,C 180,E1 -17875.095,E2 -17875.095} C_VEL
LIN {X 0,Y 270.186,Z 83.827,A -85,B 0,C 180,E1 -17879.137,E2 -17879.137} C_VEL
LIN {X 0,Y 270.224,Z 83.818,A -85,B 0,C 180,E1 -17882.164,E2 -17882.164} C_VEL
LIN {X 0,Y 270.219,Z 83.826,A -85,B 0,C 180,E1 -17885.548,E2 -17885.548} C_VEL
LIN {X 0,Y 270.24,Z 83.823,A -85,B 0,C 180,E1 -17889.038,E2 -17889.038} C_VEL
LIN {X 0,Y 271.372,Z 86.829,A -85,B 0,C 180,E1 -17889.271,E2 -17889.271} C_VEL
LIN {X 0,Y 275.394,Z 95.744,A -85,B 0,C 180,E1 -17889.914,E2 -17889.914} C_VEL
LIN {X 0,Y 282.327,Z 114.885,A -85,B 0,C 180,E1 -17891.076,E2 -17891.076} C_VEL
LIN {X 0,Y 280.404,Z 190.763,A -85,B 0,C 180,E1 -17893.014,E2 -17893.014} C_VEL
LIN {X 0,Y 279.705,Z 203.765,A -85,B 0,C 180,E1 -17893.628,E2 -17893.628} C_VEL
LIN {X 0,Y 278.738,Z 216.856,A -85,B 0,C 180,E1 -17894.555,E2 -17894.555} C_VEL
LIN {X 0,Y 277.565,Z 228.669,A -85,B 0,C 180,E1 -17895.708,E2 -17895.708} C_VEL
LIN {X 0,Y 276.138,Z 240.012,A -85,B 0,C 180,E1 -17897.133,E2 -17897.133} C_VEL
LIN {X 0,Y 274.654,Z 250.247,A -85,B 0,C 180,E1 -17898.749,E2 -17898.749} C_VEL
LIN {X 0,Y 273.274,Z 258.627,A -85,B 0,C 180,E1 -17900.377,E2 -17900.377} C_VEL
LIN {X 0,Y 271.829,Z 267.696,A -85,B 0,C 180,E1 -17902.573,E2 -17902.573} C_VEL
LIN {X 0,Y 270.601,Z 275.01,A -85,B 0,C 180,E1 -17904.785,E2 -17904.785} C_VEL
LIN {X 0,Y 269.72,Z 280.874,A -85,B 0,C 180,E1 -17907.013,E2 -17907.013} C_VEL
LIN {X 0,Y 269.082,Z 285.508,A -85,B 0,C 180,E1 -17909.252,E2 -17909.252} C_VEL
LIN {X 0,Y 268.623,Z 289.055,A -85,B 0,C 180,E1 -17911.5,E2 -17911.5} C_VEL
LIN {X 0,Y 268.47,Z 290.874,A -85,B 0,C 180,E1 -17913.002,E2 -17913.002} C_VEL
LIN {X 0,Y 268.438,Z 293.096,A -85,B 0,C 180,E1 -17915.792,E2 -17915.792} C_VEL
LIN {X 0,Y 268.342,Z 293.817,A -85,B 0,C 180,E1 -17917.525,E2 -17917.525} C_VEL
LIN {X 0,Y 268.335,Z 294.014,A -85,B 0,C 180,E1 -17919.042,E2 -17919.042} C_VEL
LIN {X 0,Y 268.683,Z 293.172,A -85,B 0,C 180,E1 -17922.079,E2 -17922.079} C_VEL
LIN {X 0,Y 269.09,Z 292.166,A -85,B 0,C 180,E1 -17923.596,E2 -17923.596} C_VEL
LIN {X 0,Y 269.645,Z 290.464,A -85,B 0,C 180,E1 -17925.339,E2 -17925.339} C_VEL
LIN {X 0,Y 270.814,Z 286.518,A -85,B 0,C 180,E1 -17928.145,E2 -17928.145} C_VEL
LIN {X 0,Y 272.118,Z 282.092,A -85,B 0,C 180,E1 -17930.406,E2 -17930.406} C_VEL
LIN {X 0,Y 273.725,Z 276.436,A -85,B 0,C 180,E1 -17932.652,E2 -17932.652} C_VEL
LIN {X 0,Y 275.72,Z 269.293,A -85,B 0,C 180,E1 -17934.872,E2 -17934.872} C_VEL
LIN {X 0,Y 278.056,Z 260.352,A -85,B 0,C 180,E1 -17937.063,E2 -17937.063} C_VEL
LIN {X 0,Y 280.169,Z 251.133,A -85,B 0,C 180,E1 -17938.874,E2 -17938.874} C_VEL
LIN {X 0,Y 282.334,Z 240.822,A -85,B 0,C 180,E1 -17940.477,E2 -17940.477} C_VEL
LIN {X 0,Y 284.444,Z 229.327,A -85,B 0,C 180,E1 -17941.88,E2 -17941.88} C_VEL
LIN {X 0,Y 286.204,Z 217.909,A -85,B 0,C 180,E1 -17942.954,E2 -17942.954} C_VEL
LIN {X 0,Y 287.404,Z 206.816,A -85,B 0,C 180,E1 -17943.755,E2 -17943.755} C_VEL
LIN {X 0,Y 288.534,Z 193.765,A -85,B 0,C 180,E1 -17944.388,E2 -17944.388} C_VEL
LIN {X 0,Y 289.313,Z 174.985,A -85,B 0,C 180,E1 -17944.916,E2 -17944.916} C_VEL
LIN {X 0,Y 290.867,Z 125.724,A -85,B 0,C 180,E1 -17946.133,E2 -17946.133} C_VEL
LIN {X 0,Y 283.481,Z 109.152,A -85,B 0,C 180,E1 -17947.579,E2 -17947.579} C_VEL
LIN {X 0,Y 275.868,Z 94.536,A -85,B 0,C 180,E1 -17949.103,E2 -17949.103} C_VEL
LIN {X 0,Y 271.804,Z 87.518,A -85,B 0,C 180,E1 -17949.939,E2 -17949.939} C_VEL
LIN {X 0,Y 270.508,Z 85.24,A -85,B 0,C 180,E1 -17950.214,E2 -17950.214} C_VEL
LIN {X 0,Y 270.253,Z 84.361,A -85,B 0,C 180,E1 -17950.35,E2 -17950.35} C_VEL
LIN {X 0,Y 270.146,Z 83.836,A -85,B 0,C 180,E1 -17950.735,E2 -17950.735} C_VEL
LIN {X 0,Y 270.131,Z 83.817,A -85,B 0,C 180,E1 -17954.625,E2 -17954.625} C_VEL
LIN {X 0,Y 270.154,Z 83.835,A -85,B 0,C 180,E1 -17957.437,E2 -17957.437} C_VEL
LIN {X 0,Y 270.195,Z 83.823,A -85,B 0,C 180,E1 -17961.371,E2 -17961.371} C_VEL
LIN {X 0,Y 270.2,Z 83.821,A -85,B 0,C 180,E1 -17965.094,E2 -17965.094} C_VEL
LIN {X 0,Y 270.174,Z 83.824,A -85,B 0,C 180,E1 -17969.141,E2 -17969.141} C_VEL
LIN {X 0,Y 270.201,Z 83.818,A -85,B 0,C 180,E1 -17972.173,E2 -17972.173} C_VEL
LIN {X 0,Y 270.23,Z 83.822,A -85,B 0,C 180,E1 -17975.543,E2 -17975.543} C_VEL
LIN {X 0,Y 270.19,Z 83.82,A -85,B 0,C 180,E1 -17978.276,E2 -17978.276} C_VEL
LIN {X 0,Y 269.587,Z 83.905,A -85,B 0,C 180,E1 -17979.52,E2 -17979.52} C_VEL
LIN {X 0,Y 266.834,Z 84.252,A -85,B 0,C 180,E1 -17981.55,E2 -17981.55} C_VEL
LIN {X 0,Y 264.452,Z 84.546,A -85,B 0,C 180,E1 -17983.199,E2 -17983.199} C_VEL
LIN {X 0,Y 263.401,Z 84.673,A -85,B 0,C 180,E1 -17984.476,E2 -17984.476} C_VEL
LIN {X 0,Y 263.301,Z 84.683,A -85,B 0,C 180,E1 -17984.909,E2 -17984.909} C_VEL
LIN {X 0,Y 263.349,Z 84.672,A -85,B 0,C 180,E1 -17989.233,E2 -17989.233} C_VEL
LIN {X 0,Y 263.528,Z 84.651,A -85,B 0,C 180,E1 -17992.337,E2 -17992.337} C_VEL
LIN {X 0,Y 263.738,Z 84.623,A -85,B 0,C 180,E1 -17998.473,E2 -17998.473} C_VEL
LIN {X 0,Y 263.742,Z 84.626,A -85,B 0,C 180,E1 -18001.527,E2 -18001.527} C_VEL
LIN {X 0,Y 263.529,Z 84.651,A -85,B 0,C 180,E1 -18007.663,E2 -18007.663} C_VEL
LIN {X 0,Y 263.352,Z 84.669,A -85,B 0,C 180,E1 -18010.766,E2 -18010.766} C_VEL
LIN {X 0,Y 263.326,Z 84.679,A -85,B 0,C 180,E1 -18015.479,E2 -18015.479} C_VEL
LIN {X 0,Y 263.265,Z 84.689,A -85,B 0,C 180,E1 -18020.306,E2 -18020.306} C_VEL
LIN {X 0,Y 263.211,Z 84.696,A -85,B 0,C 180,E1 -18025.291,E2 -18025.291} C_VEL
LIN {X 0,Y 263.182,Z 84.702,A -85,B 0,C 180,E1 -18028.729,E2 -18028.729} C_VEL
LIN {X 0,Y 263.135,Z 84.705,A -85,B 0,C 180,E1 -18032.288,E2 -18032.288} C_VEL
LIN {X 0,Y 263.187,Z 84.67,A -85,B 0,C 180,E1 -18036.763,E2 -18036.763} C_VEL
LIN {X 0,Y 263.126,Z 84.706,A -85,B 0,C 180,E1 -18041.593,E2 -18041.593} C_VEL
LIN {X 0,Y 263.124,Z 84.709,A -85,B 0,C 180,E1 -18043.984,E2 -18043.984} C_VEL
LIN {X 0,Y 263.141,Z 84.765,A -85,B 0,C 180,E1 -18048.592,E2 -18048.592} C_VEL
LIN {X 0,Y 265.655,Z 93.891,A -85,B 0,C 180,E1 -18052.529,E2 -18052.529} C_VEL
LIN {X 0,Y 268.056,Z 103.794,A -85,B 0,C 180,E1 -18056.428,E2 -18056.428} C_VEL
LIN {X 0,Y 276.979,Z 122.907,A -85,B 0,C 180,E1 -18058.364,E2 -18058.364} C_VEL
LIN {X 0,Y 278.714,Z 127.47,A -85,B 0,C 180,E1 -18058.746,E2 -18058.746} C_VEL
LIN {X 0,Y 283.234,Z 154.058,A -85,B 0,C 180,E1 -18060.147,E2 -18060.147} C_VEL
LIN {X 0,Y 283.802,Z 159.146,A -85,B 0,C 180,E1 -18060.37,E2 -18060.37} C_VEL
LIN {X 0,Y 281.78,Z 213.687,A -85,B 0,C 180,E1 -18061.763,E2 -18061.763} C_VEL
LIN {X 0,Y 280.534,Z 227.434,A -85,B 0,C 180,E1 -18062.389,E2 -18062.389} C_VEL
LIN {X 0,Y 278.829,Z 239.8,A -85,B 0,C 180,E1 -18063.221,E2 -18063.221} C_VEL
LIN {X 0,Y 276.93,Z 250.857,A -85,B 0,C 180,E1 -18064.239,E2 -18064.239} C_VEL
LIN {X 0,Y 274.546,Z 262.395,A -85,B 0,C 180,E1 -18065.62,E2 -18065.62} C_VEL
LIN {X 0,Y 272.112,Z 272.798,A -85,B 0,C 180,E1 -18067.206,E2 -18067.206} C_VEL
LIN {X 0,Y 269.706,Z 282.184,A -85,B 0,C 180,E1 -18069.004,E2 -18069.004} C_VEL
LIN {X 0,Y 267.371,Z 290.983,A -85,B 0,C 180,E1 -18071.135,E2 -18071.135} C_VEL
LIN {X 0,Y 265.324,Z 298.596,A -85,B 0,C 180,E1 -18073.456,E2 -18073.456} C_VEL
LIN {X 0,Y 263.948,Z 303.59,A -85,B 0,C 180,E1 -18075.347,E2 -18075.347} C_VEL
LIN {X 0,Y 262.602,Z 308.457,A -85,B 0,C 180,E1 -18077.637,E2 -18077.637} C_VEL
LIN {X 0,Y 261.789,Z 312.223,A -85,B 0,C 180,E1 -18079.95,E2 -18079.95} C_VEL
LIN {X 0,Y 261.311,Z 314.986,A -85,B 0,C 180,E1 -18082.271,E2 -18082.271} C_VEL
LIN {X 0,Y 261.093,Z 317.232,A -85,B 0,C 180,E1 -18085.368,E2 -18085.368} C_VEL
LIN {X 0,Y 261.145,Z 317.743,A -85,B 0,C 180,E1 -18086.914,E2 -18086.914} C_VEL
LIN {X 0,Y 261.195,Z 317.837,A -85,B 0,C 180,E1 -18088.458,E2 -18088.458} C_VEL
LIN {X 0,Y 261.248,Z 317.543,A -85,B 0,C 180,E1 -18090,E2 -18090} C_VEL
LIN {X 0,Y 261.214,Z 316.854,A -85,B 0,C 180,E1 -18091.541,E2 -18091.541} C_VEL
LIN {X 0,Y 261.194,Z 315.744,A -85,B 0,C 180,E1 -18093.084,E2 -18093.084} C_VEL
LIN {X 0,Y 261.123,Z 313.478,A -85,B 0,C 180,E1 -18095.23,E2 -18095.23} C_VEL
LIN {X 0,Y 261.299,Z 309.767,A -85,B 0,C 180,E1 -18097.728,E2 -18097.728} C_VEL
LIN {X 0,Y 261.679,Z 305.158,A -85,B 0,C 180,E1 -18100.053,E2 -18100.053} C_VEL
LIN {X 0,Y 262.533,Z 298.163,A -85,B 0,C 180,E1 -18102.759,E2 -18102.759} C_VEL
LIN {X 0,Y 263.698,Z 290.589,A -85,B 0,C 180,E1 -18105.061,E2 -18105.061} C_VEL
LIN {X 0,Y 265.022,Z 282.86,A -85,B 0,C 180,E1 -18106.96,E2 -18106.96} C_VEL
LIN {X 0,Y 266.249,Z 273.411,A -85,B 0,C 180,E1 -18108.865,E2 -18108.865} C_VEL
LIN {X 0,Y 268.026,Z 262.945,A -85,B 0,C 180,E1 -18110.53,E2 -18110.53} C_VEL
LIN {X 0,Y 269.708,Z 251.302,A -85,B 0,C 180,E1 -18111.998,E2 -18111.998} C_VEL
LIN {X 0,Y 271.255,Z 238.988,A -85,B 0,C 180,E1 -18113.172,E2 -18113.172} C_VEL
LIN {X 0,Y 272.629,Z 225.253,A -85,B 0,C 180,E1 -18114.106,E2 -18114.106} C_VEL
LIN {X 0,Y 273.393,Z 212.546,A -85,B 0,C 180,E1 -18114.676,E2 -18114.676} C_VEL
LIN {X 0,Y 274.91,Z 153.819,A -85,B 0,C 180,E1 -18116.203,E2 -18116.203} C_VEL
LIN {X 0,Y 270.901,Z 121.77,A -85,B 0,C 180,E1 -18117.473,E2 -18117.473} C_VEL
LIN {X 0,Y 268.842,Z 109.09,A -85,B 0,C 180,E1 -18118.036,E2 -18118.036} C_VEL
LIN {X 0,Y 267.41,Z 104.64,A -85,B 0,C 180,E1 -18118.327,E2 -18118.327} C_VEL
LIN {X 0,Y 265.228,Z 93.771,A -85,B 0,C 180,E1 -18122.012,E2 -18122.012} C_VEL
LIN {X 0,Y 263.215,Z 84.705,A -85,B 0,C 180,E1 -18125.282,E2 -18125.282} C_VEL
LIN {X 0,Y 263.135,Z 84.71,A -85,B 0,C 180,E1 -18129.236,E2 -18129.236} C_VEL
LIN {X 0,Y 263.123,Z 84.71,A -85,B 0,C 180,E1 -18131.893,E2 -18131.893} C_VEL
LIN {X 0,Y 263.104,Z 84.711,A -85,B 0,C 180,E1 -18136.155,E2 -18136.155} C_VEL
LIN {X 0,Y 263.104,Z 84.702,A -85,B 0,C 180,E1 -18140.127,E2 -18140.127} C_VEL
LIN {X 0,Y 263.162,Z 84.701,A -85,B 0,C 180,E1 -18144.018,E2 -18144.018} C_VEL
LIN {X 0,Y 263.132,Z 84.707,A -85,B 0,C 180,E1 -18147.712,E2 -18147.712} C_VEL
LIN {X 0,Y 263.2,Z 84.696,A -85,B 0,C 180,E1 -18151.783,E2 -18151.783} C_VEL
LIN {X 0,Y 263.225,Z 84.697,A -85,B 0,C 180,E1 -18155.2,E2 -18155.2} C_VEL
LIN {X 0,Y 263.263,Z 84.682,A -85,B 0,C 180,E1 -18159.694,E2 -18159.694} C_VEL
LIN {X 0,Y 263.35,Z 84.681,A -85,B 0,C 180,E1 -18164.522,E2 -18164.522} C_VEL
LIN {X 0,Y 263.354,Z 84.675,A -85,B 0,C 180,E1 -18169.234,E2 -18169.234} C_VEL
LIN {X 0,Y 263.557,Z 84.657,A -85,B 0,C 180,E1 -18172.338,E2 -18172.338} C_VEL
LIN {X 0,Y 263.748,Z 84.63,A -85,B 0,C 180,E1 -18178.473,E2 -18178.473} C_VEL
LIN {X 0,Y 263.748,Z 84.63,A -85,B 0,C 180,E1 -18181.527,E2 -18181.527} C_VEL
LIN {X 0,Y 263.533,Z 84.656,A -85,B 0,C 180,E1 -18187.663,E2 -18187.663} C_VEL
LIN {X 0,Y 263.349,Z 84.676,A -85,B 0,C 180,E1 -18190.767,E2 -18190.767} C_VEL
LIN {X 0,Y 263.351,Z 84.677,A -85,B 0,C 180,E1 -18195.478,E2 -18195.478} C_VEL
LIN {X 0,Y 263.264,Z 84.683,A -85,B 0,C 180,E1 -18200.307,E2 -18200.307} C_VEL
LIN {X 0,Y 263.208,Z 84.7,A -85,B 0,C 180,E1 -18205.292,E2 -18205.292} C_VEL
LIN {X 0,Y 263.166,Z 84.702,A -85,B 0,C 180,E1 -18208.732,E2 -18208.732} C_VEL
LIN {X 0,Y 263.133,Z 84.706,A -85,B 0,C 180,E1 -18212.289,E2 -18212.289} C_VEL
LIN {X 0,Y 263.18,Z 84.704,A -85,B 0,C 180,E1 -18216.763,E2 -18216.763} C_VEL
LIN {X 0,Y 263.092,Z 84.712,A -85,B 0,C 180,E1 -18219.876,E2 -18219.876} C_VEL
LIN {X 0,Y 263.098,Z 84.711,A -85,B 0,C 180,E1 -18223.99,E2 -18223.99} C_VEL
LIN {X 0,Y 263.124,Z 84.71,A -85,B 0,C 180,E1 -18228.408,E2 -18228.408} C_VEL
LIN {X 0,Y 263.158,Z 84.705,A -85,B 0,C 180,E1 -18232.103,E2 -18232.103} C_VEL
LIN {X 0,Y 263.153,Z 84.705,A -85,B 0,C 180,E1 -18235.886,E2 -18235.886} C_VEL
LIN {X 0,Y 263.128,Z 84.706,A -85,B 0,C 180,E1 -18239.504,E2 -18239.504} C_VEL
LIN {X 0,Y 263.141,Z 84.706,A -85,B 0,C 180,E1 -18242.997,E2 -18242.997} C_VEL
LIN {X 0,Y 263.141,Z 84.709,A -85,B 0,C 180,E1 -18246.383,E2 -18246.383} C_VEL
LIN {X 0,Y 263.161,Z 84.706,A -85,B 0,C 180,E1 -18248.364,E2 -18248.364} C_VEL
LIN {X 0,Y 264.251,Z 87.69,A -85,B 0,C 180,E1 -18248.571,E2 -18248.571} C_VEL
LIN {X 0,Y 269.097,Z 97.92,A -85,B 0,C 180,E1 -18249.365,E2 -18249.365} C_VEL
LIN {X 0,Y 275.806,Z 116.432,A -85,B 0,C 180,E1 -18250.533,E2 -18250.533} C_VEL
LIN {X 0,Y 273.769,Z 191.437,A -85,B 0,C 180,E1 -18252.493,E2 -18252.493} C_VEL
LIN {X 0,Y 273.015,Z 205.071,A -85,B 0,C 180,E1 -18253.166,E2 -18253.166} C_VEL
LIN {X 0,Y 272.057,Z 217.338,A -85,B 0,C 180,E1 -18254.07,E2 -18254.07} C_VEL
LIN {X 0,Y 270.748,Z 229.895,A -85,B 0,C 180,E1 -18255.34,E2 -18255.34} C_VEL
LIN {X 0,Y 269.276,Z 241.072,A -85,B 0,C 180,E1 -18256.799,E2 -18256.799} C_VEL
LIN {X 0,Y 267.742,Z 251.155,A -85,B 0,C 180,E1 -18258.455,E2 -18258.455} C_VEL
LIN {X 0,Y 266.033,Z 261.049,A -85,B 0,C 180,E1 -18260.497,E2 -18260.497} C_VEL
LIN {X 0,Y 264.584,Z 269.754,A -85,B 0,C 180,E1 -18262.752,E2 -18262.752} C_VEL
LIN {X 0,Y 263.401,Z 276.718,A -85,B 0,C 180,E1 -18265.026,E2 -18265.026} C_VEL
LIN {X 0,Y 262.4,Z 283.088,A -85,B 0,C 180,E1 -18267.698,E2 -18267.698} C_VEL
LIN {X 0,Y 261.861,Z 287.29,A -85,B 0,C 180,E1 -18270,E2 -18270} C_VEL
LIN {X 0,Y 261.525,Z 289.53,A -85,B 0,C 180,E1 -18271.54,E2 -18271.54} C_VEL
LIN {X 0,Y 261.394,Z 291.3,A -85,B 0,C 180,E1 -18273.083,E2 -18273.083} C_VEL
LIN {X 0,Y 261.366,Z 293.385,A -85,B 0,C 180,E1 -18275.777,E2 -18275.777} C_VEL
LIN {X 0,Y 261.257,Z 294.174,A -85,B 0,C 180,E1 -18277.73,E2 -18277.73} C_VEL
LIN {X 0,Y 261.251,Z 294.326,A -85,B 0,C 180,E1 -18279.289,E2 -18279.289} C_VEL
LIN {X 0,Y 261.683,Z 293.436,A -85,B 0,C 180,E1 -18282.408,E2 -18282.408} C_VEL
LIN {X 0,Y 262.092,Z 292.406,A -85,B 0,C 180,E1 -18283.966,E2 -18283.966} C_VEL
LIN {X 0,Y 262.639,Z 290.877,A -85,B 0,C 180,E1 -18285.562,E2 -18285.562} C_VEL
LIN {X 0,Y 263.572,Z 287.898,A -85,B 0,C 180,E1 -18287.857,E2 -18287.857} C_VEL
LIN {X 0,Y 264.828,Z 283.796,A -85,B 0,C 180,E1 -18290.182,E2 -18290.182} C_VEL
LIN {X 0,Y 266.621,Z 277.944,A -85,B 0,C 180,E1 -18292.692,E2 -18292.692} C_VEL
LIN {X 0,Y 268.828,Z 270.563,A -85,B 0,C 180,E1 -18295.14,E2 -18295.14} C_VEL
LIN {X 0,Y 271.216,Z 261.843,A -85,B 0,C 180,E1 -18297.385,E2 -18297.385} C_VEL
LIN {X 0,Y 273.643,Z 251.875,A -85,B 0,C 180,E1 -18299.419,E2 -18299.419} C_VEL
LIN {X 0,Y 275.589,Z 242.942,A -85,B 0,C 180,E1 -18300.879,E2 -18300.879} C_VEL
LIN {X 0,Y 277.802,Z 231.93,A -85,B 0,C 180,E1 -18302.306,E2 -18302.306} C_VEL
LIN {X 0,Y 279.826,Z 219.515,A -85,B 0,C 180,E1 -18303.542,E2 -18303.542} C_VEL
LIN {X 0,Y 281.243,Z 207.463,A -85,B 0,C 180,E1 -18304.447,E2 -18304.447} C_VEL
LIN {X 0,Y 282.423,Z 194.626,A -85,B 0,C 180,E1 -18305.09,E2 -18305.09} C_VEL
LIN {X 0,Y 283.163,Z 177.969,A -85,B 0,C 180,E1 -18305.583,E2 -18305.583} C_VEL
LIN {X 0,Y 284.873,Z 127.801,A -85,B 0,C 180,E1 -18306.839,E2 -18306.839} C_VEL
LIN {X 0,Y 277.265,Z 110.851,A -85,B 0,C 180,E1 -18308.392,E2 -18308.392} C_VEL
LIN {X 0,Y 269.604,Z 96.276,A -85,B 0,C 180,E1 -18309.998,E2 -18309.998} C_VEL
LIN {X 0,Y 266.772,Z 91.647,A -85,B 0,C 180,E1 -18310.598,E2 -18310.598} C_VEL
LIN {X 0,Y 265.027,Z 88.75,A -85,B 0,C 180,E1 -18310.979,E2 -18310.979} C_VEL
LIN {X 0,Y 263.428,Z 86.16,A -85,B 0,C 180,E1 -18311.332,E2 -18311.332} C_VEL
LIN {X 0,Y 263.123,Z 84.877,A -85,B 0,C 180,E1 -18311.448,E2 -18311.448} C_VEL
LIN {X 0,Y 263.079,Z 84.699,A -85,B 0,C 180,E1 -18313.994,E2 -18313.994} C_VEL
LIN {X 0,Y 263.083,Z 84.709,A -85,B 0,C 180,E1 -18318.418,E2 -18318.418} C_VEL
LIN {X 0,Y 263.133,Z 84.705,A -85,B 0,C 180,E1 -18322.098,E2 -18322.098} C_VEL
LIN {X 0,Y 263.155,Z 84.704,A -85,B 0,C 180,E1 -18325.885,E2 -18325.885} C_VEL
LIN {X 0,Y 263.113,Z 84.706,A -85,B 0,C 180,E1 -18329.501,E2 -18329.501} C_VEL
LIN {X 0,Y 263.132,Z 84.698,A -85,B 0,C 180,E1 -18332.995,E2 -18332.995} C_VEL
LIN {X 0,Y 263.148,Z 84.698,A -85,B 0,C 180,E1 -18336.383,E2 -18336.383} C_VEL
LIN {X 0,Y 263.247,Z 84.694,A -85,B 0,C 180,E1 -18339.692,E2 -18339.692} C_VEL
LIN {X 0,Y 263.327,Z 84.682,A -85,B 0,C 180,E1 -18344.52,E2 -18344.52} C_VEL
LIN {X 0,Y 263.301,Z 84.683,A -85,B 0,C 180,E1 -18344.909,E2 -18344.909} C_VEL
LIN {X 0,Y 262.605,Z 84.77,A -85,B 0,C 180,E1 -18346.185,E2 -18346.185} C_VEL
LIN {X 0,Y 259.796,Z 85.118,A -85,B 0,C 180,E1 -18348.269,E2 -18348.269} C_VEL
LIN {X 0,Y 257.463,Z 85.411,A -85,B 0,C 180,E1 -18349.963,E2 -18349.963} C_VEL
LIN {X 0,Y 256.503,Z 85.533,A -85,B 0,C 180,E1 -18351.275,E2 -18351.275} C_VEL
LIN {X 0,Y 256.444,Z 85.535,A -85,B 0,C 180,E1 -18351.718,E2 -18351.718} C_VEL
LIN {X 0,Y 256.458,Z 85.522,A -85,B 0,C 180,E1 -18353.706,E2 -18353.706} C_VEL
LIN {X 0,Y 256.701,Z 85.5,A -85,B 0,C 180,E1 -18358.431,E2 -18358.431} C_VEL
LIN {X 0,Y 256.703,Z 85.503,A -85,B 0,C 180,E1 -18361.568,E2 -18361.568} C_VEL
LIN {X 0,Y 256.458,Z 85.522,A -85,B 0,C 180,E1 -18366.293,E2 -18366.293} C_VEL
LIN {X 0,Y 256.43,Z 85.542,A -85,B 0,C 180,E1 -18369.465,E2 -18369.465} C_VEL
LIN {X 0,Y 256.241,Z 85.565,A -85,B 0,C 180,E1 -18374.291,E2 -18374.291} C_VEL
LIN {X 0,Y 256.186,Z 85.558,A -85,B 0,C 180,E1 -18377.563,E2 -18377.563} C_VEL
LIN {X 0,Y 256.16,Z 85.569,A -85,B 0,C 180,E1 -18381.119,E2 -18381.119} C_VEL
LIN {X 0,Y 256.191,Z 85.572,A -85,B 0,C 180,E1 -18385.138,E2 -18385.138} C_VEL
LIN {X 0,Y 256.116,Z 85.58,A -85,B 0,C 180,E1 -18389.599,E2 -18389.599} C_VEL
LIN {X 0,Y 256.07,Z 85.587,A -85,B 0,C 180,E1 -18393.292,E2 -18393.292} C_VEL
LIN {X 0,Y 256.118,Z 85.552,A -85,B 0,C 180,E1 -18397.271,E2 -18397.271} C_VEL
LIN {X 0,Y 256.056,Z 85.585,A -85,B 0,C 180,E1 -18401.203,E2 -18401.203} C_VEL
LIN {X 0,Y 256.046,Z 85.587,A -85,B 0,C 180,E1 -18405.533,E2 -18405.533} C_VEL
LIN {X 0,Y 256.073,Z 85.685,A -85,B 0,C 180,E1 -18407.575,E2 -18407.575} C_VEL
LIN {X 0,Y 258.384,Z 93.836,A -85,B 0,C 180,E1 -18411.273,E2 -18411.273} C_VEL
LIN {X 0,Y 260.312,Z 101.564,A -85,B 0,C 180,E1 -18414.515,E2 -18414.515} C_VEL
LIN {X 0,Y 260.757,Z 103.418,A -85,B 0,C 180,E1 -18415.228,E2 -18415.228} C_VEL
LIN {X 0,Y 268.113,Z 118.581,A -85,B 0,C 180,E1 -18416.918,E2 -18416.918} C_VEL
LIN {X 0,Y 272.983,Z 129.603,A -85,B 0,C 180,E1 -18417.999,E2 -18417.999} C_VEL
LIN {X 0,Y 277.354,Z 155.733,A -85,B 0,C 180,E1 -18419.42,E2 -18419.42} C_VEL
LIN {X 0,Y 277.791,Z 159.792,A -85,B 0,C 180,E1 -18419.602,E2 -18419.602} C_VEL
LIN {X 0,Y 275.733,Z 213.337,A -85,B 0,C 180,E1 -18420.997,E2 -18420.997} C_VEL
LIN {X 0,Y 274.488,Z 226.864,A -85,B 0,C 180,E1 -18421.622,E2 -18421.622} C_VEL
LIN {X 0,Y 272.705,Z 239.306,A -85,B 0,C 180,E1 -18422.465,E2 -18422.465} C_VEL
LIN {X 0,Y 270.56,Z 251.197,A -85,B 0,C 180,E1 -18423.587,E2 -18423.587} C_VEL
LIN {X 0,Y 268.112,Z 262.613,A -85,B 0,C 180,E1 -18424.995,E2 -18424.995} C_VEL
LIN {X 0,Y 265.605,Z 272.923,A -85,B 0,C 180,E1 -18426.615,E2 -18426.615} C_VEL
LIN {X 0,Y 263.082,Z 282.204,A -85,B 0,C 180,E1 -18428.449,E2 -18428.449} C_VEL
LIN {X 0,Y 260.941,Z 289.866,A -85,B 0,C 180,E1 -18430.326,E2 -18430.326} C_VEL
LIN {X 0,Y 258.832,Z 297.387,A -85,B 0,C 180,E1 -18432.621,E2 -18432.621} C_VEL
LIN {X 0,Y 257.068,Z 303.457,A -85,B 0,C 180,E1 -18434.946,E2 -18434.946} C_VEL
LIN {X 0,Y 255.628,Z 308.283,A -85,B 0,C 180,E1 -18437.294,E2 -18437.294} C_VEL
LIN {X 0,Y 254.766,Z 312.011,A -85,B 0,C 180,E1 -18439.67,E2 -18439.67} C_VEL
LIN {X 0,Y 254.249,Z 314.739,A -85,B 0,C 180,E1 -18442.055,E2 -18442.055} C_VEL
LIN {X 0,Y 254.013,Z 316.95,A -85,B 0,C 180,E1 -18445.238,E2 -18445.238} C_VEL
LIN {X 0,Y 254.056,Z 317.43,A -85,B 0,C 180,E1 -18446.828,E2 -18446.828} C_VEL
LIN {X 0,Y 254.119,Z 317.509,A -85,B 0,C 180,E1 -18448.415,E2 -18448.415} C_VEL
LIN {X 0,Y 254.17,Z 317.199,A -85,B 0,C 180,E1 -18450,E2 -18450} C_VEL
LIN {X 0,Y 254.139,Z 316.493,A -85,B 0,C 180,E1 -18451.584,E2 -18451.584} C_VEL
LIN {X 0,Y 254.103,Z 315.349,A -85,B 0,C 180,E1 -18453.171,E2 -18453.171} C_VEL
LIN {X 0,Y 254.029,Z 313.334,A -85,B 0,C 180,E1 -18455.14,E2 -18455.14} C_VEL
LIN {X 0,Y 254.237,Z 309.308,A -85,B 0,C 180,E1 -18457.944,E2 -18457.944} C_VEL
LIN {X 0,Y 254.657,Z 304.655,A -85,B 0,C 180,E1 -18460.334,E2 -18460.334} C_VEL
LIN {X 0,Y 255.573,Z 297.609,A -85,B 0,C 180,E1 -18463.112,E2 -18463.112} C_VEL
LIN {X 0,Y 256.796,Z 289.983,A -85,B 0,C 180,E1 -18465.476,E2 -18465.476} C_VEL
LIN {X 0,Y 258.164,Z 282.192,A -85,B 0,C 180,E1 -18467.424,E2 -18467.424} C_VEL
LIN {X 0,Y 259.499,Z 272.639,A -85,B 0,C 180,E1 -18469.376,E2 -18469.376} C_VEL
LIN {X 0,Y 261.362,Z 262.08,A -85,B 0,C 180,E1 -18471.078,E2 -18471.078} C_VEL
LIN {X 0,Y 263.114,Z 250.308,A -85,B 0,C 180,E1 -18472.579,E2 -18472.579} C_VEL
LIN {X 0,Y 264.702,Z 237.712,A -85,B 0,C 180,E1 -18473.78,E2 -18473.78} C_VEL
LIN {X 0,Y 266.065,Z 224.413,A -85,B 0,C 180,E1 -18474.688,E2 -18474.688} C_VEL
LIN {X 0,Y 266.849,Z 211.853,A -85,B 0,C 180,E1 -18475.249,E2 -18475.249} C_VEL
LIN {X 0,Y 268.325,Z 153.772,A -85,B 0,C 180,E1 -18476.8,E2 -18476.8} C_VEL
LIN {X 0,Y 264.572,Z 123.702,A -85,B 0,C 180,E1 -18478.033,E2 -18478.033} C_VEL
LIN {X 0,Y 262.638,Z 111.313,A -85,B 0,C 180,E1 -18478.594,E2 -18478.594} C_VEL
LIN {X 0,Y 260.137,Z 104.257,A -85,B 0,C 180,E1 -18479.097,E2 -18479.097} C_VEL
LIN {X 0,Y 258.181,Z 94.702,A -85,B 0,C 180,E1 -18482.45,E2 -18482.45} C_VEL
LIN {X 0,Y 256.255,Z 86.043,A -85,B 0,C 180,E1 -18485.647,E2 -18485.647} C_VEL
LIN {X 0,Y 256.151,Z 85.584,A -85,B 0,C 180,E1 -18485.906,E2 -18485.906} C_VEL
LIN {X 0,Y 256.071,Z 85.589,A -85,B 0,C 180,E1 -18489.783,E2 -18489.783} C_VEL
LIN {X 0,Y 256.06,Z 85.59,A -85,B 0,C 180,E1 -18493.327,E2 -18493.327} C_VEL
LIN {X 0,Y 256.068,Z 85.588,A -85,B 0,C 180,E1 -18497.819,E2 -18497.819} C_VEL
LIN {X 0,Y 256.07,Z 85.573,A -85,B 0,C 180,E1 -18500.858,E2 -18500.858} C_VEL
LIN {X 0,Y 256.129,Z 85.57,A -85,B 0,C 180,E1 -18502.867,E2 -18502.867} C_VEL
LIN {X 0,Y 256.066,Z 85.587,A -85,B 0,C 180,E1 -18506.707,E2 -18506.707} C_VEL
LIN {X 0,Y 256.113,Z 85.581,A -85,B 0,C 180,E1 -18510.4,E2 -18510.4} C_VEL
LIN {X 0,Y 256.188,Z 85.571,A -85,B 0,C 180,E1 -18514.861,E2 -18514.861} C_VEL
LIN {X 0,Y 256.166,Z 85.567,A -85,B 0,C 180,E1 -18519.105,E2 -18519.105} C_VEL
LIN {X 0,Y 256.299,Z 85.558,A -85,B 0,C 180,E1 -18524.085,E2 -18524.085} C_VEL
LIN {X 0,Y 256.294,Z 85.547,A -85,B 0,C 180,E1 -18527.328,E2 -18527.328} C_VEL
LIN {X 0,Y 256.515,Z 85.533,A -85,B 0,C 180,E1 -18532.127,E2 -18532.127} C_VEL
LIN {X 0,Y 256.494,Z 85.527,A -85,B 0,C 180,E1 -18536.859,E2 -18536.859} C_VEL
LIN {X 0,Y 256.756,Z 85.503,A -85,B 0,C 180,E1 -18540,E2 -18540} C_VEL
LIN {X 0,Y 256.492,Z 85.529,A -85,B 0,C 180,E1 -18543.142,E2 -18543.142} C_VEL
LIN {X 0,Y 256.495,Z 85.534,A -85,B 0,C 180,E1 -18547.875,E2 -18547.875} C_VEL
LIN {X 0,Y 256.291,Z 85.555,A -85,B 0,C 180,E1 -18551.067,E2 -18551.067} C_VEL
LIN {X 0,Y 256.3,Z 85.557,A -85,B 0,C 180,E1 -18555.915,E2 -18555.915} C_VEL
LIN {X 0,Y 256.167,Z 85.567,A -85,B 0,C 180,E1 -18560.896,E2 -18560.896} C_VEL
LIN {X 0,Y 256.188,Z 85.573,A -85,B 0,C 180,E1 -18565.139,E2 -18565.139} C_VEL
LIN {X 0,Y 256.104,Z 85.582,A -85,B 0,C 180,E1 -18569.602,E2 -18569.602} C_VEL
LIN {X 0,Y 256.068,Z 85.588,A -85,B 0,C 180,E1 -18573.293,E2 -18573.293} C_VEL
LIN {X 0,Y 256.113,Z 85.582,A -85,B 0,C 180,E1 -18577.271,E2 -18577.271} C_VEL
LIN {X 0,Y 256.019,Z 85.593,A -85,B 0,C 180,E1 -18581.211,E2 -18581.211} C_VEL
LIN {X 0,Y 256.04,Z 85.59,A -85,B 0,C 180,E1 -18585.535,E2 -18585.535} C_VEL
LIN {X 0,Y 256.054,Z 85.591,A -85,B 0,C 180,E1 -18588.797,E2 -18588.797} C_VEL
LIN {X 0,Y 256.128,Z 85.581,A -85,B 0,C 180,E1 -18592.868,E2 -18592.868} C_VEL
LIN {X 0,Y 256.068,Z 85.585,A -85,B 0,C 180,E1 -18596.708,E2 -18596.708} C_VEL
LIN {X 0,Y 256.056,Z 85.58,A -85,B 0,C 180,E1 -18600.394,E2 -18600.394} C_VEL
LIN {X 0,Y 256.085,Z 85.587,A -85,B 0,C 180,E1 -18603.954,E2 -18603.954} C_VEL
LIN {X 0,Y 256.076,Z 85.589,A -85,B 0,C 180,E1 -18607.59,E2 -18607.59} C_VEL
LIN {X 0,Y 257.24,Z 88.657,A -85,B 0,C 180,E1 -18607.843,E2 -18607.843} C_VEL
LIN {X 0,Y 262.819,Z 100.199,A -85,B 0,C 180,E1 -18608.792,E2 -18608.792} C_VEL
LIN {X 0,Y 269.312,Z 117.931,A -85,B 0,C 180,E1 -18609.963,E2 -18609.963} C_VEL
LIN {X 0,Y 267.25,Z 190.959,A -85,B 0,C 180,E1 -18611.903,E2 -18611.903} C_VEL
LIN {X 0,Y 266.512,Z 204.103,A -85,B 0,C 180,E1 -18612.545,E2 -18612.545} C_VEL
LIN {X 0,Y 265.474,Z 216.733,A -85,B 0,C 180,E1 -18613.466,E2 -18613.466} C_VEL
LIN {X 0,Y 264.338,Z 227.969,A -85,B 0,C 180,E1 -18614.582,E2 -18614.582} C_VEL
LIN {X 0,Y 262.814,Z 239.56,A -85,B 0,C 180,E1 -18616.074,E2 -18616.074} C_VEL
LIN {X 0,Y 261.179,Z 249.987,A -85,B 0,C 180,E1 -18617.766,E2 -18617.766} C_VEL
LIN {X 0,Y 259.696,Z 258.518,A -85,B 0,C 180,E1 -18619.475,E2 -18619.475} C_VEL
LIN {X 0,Y 258.305,Z 266.377,A -85,B 0,C 180,E1 -18621.394,E2 -18621.394} C_VEL
LIN {X 0,Y 256.941,Z 274.071,A -85,B 0,C 180,E1 -18623.719,E2 -18623.719} C_VEL
LIN {X 0,Y 255.874,Z 280.237,A -85,B 0,C 180,E1 -18626.063,E2 -18626.063} C_VEL
LIN {X 0,Y 255.137,Z 285.139,A -85,B 0,C 180,E1 -18628.422,E2 -18628.422} C_VEL
LIN {X 0,Y 254.585,Z 288.939,A -85,B 0,C 180,E1 -18630.791,E2 -18630.791} C_VEL
LIN {X 0,Y 254.317,Z 291.724,A -85,B 0,C 180,E1 -18633.169,E2 -18633.169} C_VEL
LIN {X 0,Y 254.274,Z 293.65,A -85,B 0,C 180,E1 -18635.713,E2 -18635.713} C_VEL
LIN {X 0,Y 254.171,Z 294.522,A -85,B 0,C 180,E1 -18637.947,E2 -18637.947} C_VEL
LIN {X 0,Y 254.345,Z 294.363,A -85,B 0,C 180,E1 -18641.153,E2 -18641.153} C_VEL
LIN {X 0,Y 254.663,Z 293.702,A -85,B 0,C 180,E1 -18642.755,E2 -18642.755} C_VEL
LIN {X 0,Y 255.112,Z 292.637,A -85,B 0,C 180,E1 -18644.356,E2 -18644.356} C_VEL
LIN {X 0,Y 255.677,Z 291.116,A -85,B 0,C 180,E1 -18645.955,E2 -18645.955} C_VEL
LIN {X 0,Y 256.722,Z 288.042,A -85,B 0,C 180,E1 -18648.351,E2 -18648.351} C_VEL
LIN {X 0,Y 258.075,Z 283.886,A -85,B 0,C 180,E1 -18650.734,E2 -18650.734} C_VEL
LIN {X 0,Y 260.142,Z 277.476,A -85,B 0,C 180,E1 -18653.498,E2 -18653.498} C_VEL
LIN {X 0,Y 262.304,Z 270.513,A -85,B 0,C 180,E1 -18655.811,E2 -18655.811} C_VEL
LIN {X 0,Y 264.828,Z 261.692,A -85,B 0,C 180,E1 -18658.103,E2 -18658.103} C_VEL
LIN {X 0,Y 267.336,Z 251.622,A -85,B 0,C 180,E1 -18660.184,E2 -18660.184} C_VEL
LIN {X 0,Y 269.653,Z 241.263,A -85,B 0,C 180,E1 -18661.856,E2 -18661.856} C_VEL
LIN {X 0,Y 272.011,Z 229.729,A -85,B 0,C 180,E1 -18663.302,E2 -18663.302} C_VEL
LIN {X 0,Y 273.847,Z 218.679,A -85,B 0,C 180,E1 -18664.376,E2 -18664.376} C_VEL
LIN {X 0,Y 275.168,Z 207.636,A -85,B 0,C 180,E1 -18665.203,E2 -18665.203} C_VEL
LIN {X 0,Y 276.394,Z 194.766,A -85,B 0,C 180,E1 -18665.853,E2 -18665.853} C_VEL
LIN {X 0,Y 277.16,Z 177.506,A -85,B 0,C 180,E1 -18666.37,E2 -18666.37} C_VEL
LIN {X 0,Y 278.848,Z 129.802,A -85,B 0,C 180,E1 -18667.588,E2 -18667.588} C_VEL
LIN {X 0,Y 271.723,Z 113.856,A -85,B 0,C 180,E1 -18669.109,E2 -18669.109} C_VEL
LIN {X 0,Y 264.43,Z 99.97,A -85,B 0,C 180,E1 -18670.702,E2 -18670.702} C_VEL
LIN {X 0,Y 260.002,Z 92.914,A -85,B 0,C 180,E1 -18671.685,E2 -18671.685} C_VEL
LIN {X 0,Y 258.079,Z 89.763,A -85,B 0,C 180,E1 -18672.129,E2 -18672.129} C_VEL
LIN {X 0,Y 256.424,Z 87.255,A -85,B 0,C 180,E1 -18672.512,E2 -18672.512} C_VEL
LIN {X 0,Y 256.01,Z 85.597,A -85,B 0,C 180,E1 -18672.656,E2 -18672.656} C_VEL
LIN {X 0,Y 256.025,Z 85.591,A -85,B 0,C 180,E1 -18676.664,E2 -18676.664} C_VEL
LIN {X 0,Y 256.068,Z 85.584,A -85,B 0,C 180,E1 -18680.857,E2 -18680.857} C_VEL
LIN {X 0,Y 256.082,Z 85.579,A -85,B 0,C 180,E1 -18684.806,E2 -18684.806} C_VEL
LIN {X 0,Y 256.08,Z 85.577,A -85,B 0,C 180,E1 -18688.57,E2 -18688.57} C_VEL
LIN {X 0,Y 256.089,Z 85.575,A -85,B 0,C 180,E1 -18692.189,E2 -18692.189} C_VEL
LIN {X 0,Y 256.136,Z 85.577,A -85,B 0,C 180,E1 -18695.695,E2 -18695.695} C_VEL
LIN {X 0,Y 256.151,Z 85.576,A -85,B 0,C 180,E1 -18699.103,E2 -18699.103} C_VEL
LIN {X 0,Y 256.262,Z 85.56,A -85,B 0,C 180,E1 -18704.082,E2 -18704.082} C_VEL
LIN {X 0,Y 256.291,Z 85.548,A -85,B 0,C 180,E1 -18708.933,E2 -18708.933} C_VEL
LIN {X 0,Y 256.444,Z 85.535,A -85,B 0,C 180,E1 -18711.718,E2 -18711.718} C_VEL
LIN {X 0,Y 255.856,Z 85.609,A -85,B 0,C 180,E1 -18713.027,E2 -18713.027} C_VEL
LIN {X 0,Y 253.13,Z 85.954,A -85,B 0,C 180,E1 -18715.163,E2 -18715.163} C_VEL
LIN {X 0,Y 250.772,Z 86.248,A -85,B 0,C 180,E1 -18716.901,E2 -18716.901} C_VEL
LIN {X 0,Y 249.74,Z 86.369,A -85,B 0,C 180,E1 -18718.246,E2 -18718.246} C_VEL
LIN {X 0,Y 249.648,Z 86.375,A -85,B 0,C 180,E1 -18718.702,E2 -18718.702} C_VEL
LIN {X 0,Y 249.664,Z 86.38,A -85,B 0,C 180,E1 -18721.613,E2 -18721.613} C_VEL
LIN {X 0,Y 249.432,Z 86.398,A -85,B 0,C 180,E1 -18726.471,E2 -18726.471} C_VEL
LIN {X 0,Y 249.345,Z 86.421,A -85,B 0,C 180,E1 -18729.736,E2 -18729.736} C_VEL
LIN {X 0,Y 249.186,Z 86.443,A -85,B 0,C 180,E1 -18734.704,E2 -18734.704} C_VEL
LIN {X 0,Y 249.124,Z 86.441,A -85,B 0,C 180,E1 -18738.078,E2 -18738.078} C_VEL
LIN {X 0,Y 249.09,Z 86.445,A -85,B 0,C 180,E1 -18741.518,E2 -18741.518} C_VEL
LIN {X 0,Y 249.133,Z 86.448,A -85,B 0,C 180,E1 -18745.482,E2 -18745.482} C_VEL
LIN {X 0,Y 249.086,Z 86.459,A -85,B 0,C 180,E1 -18748.993,E2 -18748.993} C_VEL
LIN {X 0,Y 249.033,Z 86.463,A -85,B 0,C 180,E1 -18752.425,E2 -18752.425} C_VEL
LIN {X 0,Y 249.033,Z 86.431,A -85,B 0,C 180,E1 -18756.345,E2 -18756.345} C_VEL
LIN {X 0,Y 249.008,Z 86.464,A -85,B 0,C 180,E1 -18760.478,E2 -18760.478} C_VEL
LIN {X 0,Y 248.997,Z 86.469,A -85,B 0,C 180,E1 -18764.88,E2 -18764.88} C_VEL
LIN {X 0,Y 249.035,Z 86.624,A -85,B 0,C 180,E1 -18766.497,E2 -18766.497} C_VEL
LIN {X 0,Y 251.671,Z 95.887,A -85,B 0,C 180,E1 -18770.882,E2 -18770.882} C_VEL
LIN {X 0,Y 253.471,Z 102.959,A -85,B 0,C 180,E1 -18773.934,E2 -18773.934} C_VEL
LIN {X 0,Y 255.628,Z 107.278,A -85,B 0,C 180,E1 -18774.475,E2 -18774.475} C_VEL
LIN {X 0,Y 262.579,Z 121.382,A -85,B 0,C 180,E1 -18776.136,E2 -18776.136} C_VEL
LIN {X 0,Y 267.484,Z 132.655,A -85,B 0,C 180,E1 -18777.277,E2 -18777.277} C_VEL
LIN {X 0,Y 271.648,Z 158.452,A -85,B 0,C 180,E1 -18778.712,E2 -18778.712} C_VEL
LIN {X 0,Y 271.767,Z 162.473,A -85,B 0,C 180,E1 -18778.854,E2 -18778.854} C_VEL
LIN {X 0,Y 269.731,Z 213.164,A -85,B 0,C 180,E1 -18780.205,E2 -18780.205} C_VEL
LIN {X 0,Y 268.393,Z 227.062,A -85,B 0,C 180,E1 -18780.863,E2 -18780.863} C_VEL
LIN {X 0,Y 266.45,Z 239.843,A -85,B 0,C 180,E1 -18781.762,E2 -18781.762} C_VEL
LIN {X 0,Y 264.232,Z 251.537,A -85,B 0,C 180,E1 -18782.903,E2 -18782.903} C_VEL
LIN {X 0,Y 261.706,Z 262.832,A -85,B 0,C 180,E1 -18784.339,E2 -18784.339} C_VEL
LIN {X 0,Y 259.114,Z 273.035,A -85,B 0,C 180,E1 -18785.992,E2 -18785.992} C_VEL
LIN {X 0,Y 256.471,Z 282.222,A -85,B 0,C 180,E1 -18787.865,E2 -18787.865} C_VEL
LIN {X 0,Y 254.158,Z 290.096,A -85,B 0,C 180,E1 -18789.862,E2 -18789.862} C_VEL
LIN {X 0,Y 252.06,Z 297.299,A -85,B 0,C 180,E1 -18792.139,E2 -18792.139} C_VEL
LIN {X 0,Y 250.202,Z 303.324,A -85,B 0,C 180,E1 -18794.523,E2 -18794.523} C_VEL
LIN {X 0,Y 248.667,Z 308.109,A -85,B 0,C 180,E1 -18796.932,E2 -18796.932} C_VEL
LIN {X 0,Y 247.76,Z 311.8,A -85,B 0,C 180,E1 -18799.374,E2 -18799.374} C_VEL
LIN {X 0,Y 247.187,Z 314.492,A -85,B 0,C 180,E1 -18801.827,E2 -18801.827} C_VEL
LIN {X 0,Y 246.922,Z 316.663,A -85,B 0,C 180,E1 -18805.101,E2 -18805.101} C_VEL
LIN {X 0,Y 246.971,Z 317.117,A -85,B 0,C 180,E1 -18806.737,E2 -18806.737} C_VEL
LIN {X 0,Y 247.045,Z 317.181,A -85,B 0,C 180,E1 -18808.369,E2 -18808.369} C_VEL
LIN {X 0,Y 247.094,Z 316.854,A -85,B 0,C 180,E1 -18810,E2 -18810} C_VEL
LIN {X 0,Y 247.065,Z 316.129,A -85,B 0,C 180,E1 -18811.63,E2 -18811.63} C_VEL
LIN {X 0,Y 247.016,Z 314.952,A -85,B 0,C 180,E1 -18813.262,E2 -18813.262} C_VEL
LIN {X 0,Y 246.95,Z 313.148,A -85,B 0,C 180,E1 -18815.081,E2 -18815.081} C_VEL
LIN {X 0,Y 247.086,Z 310.129,A -85,B 0,C 180,E1 -18817.353,E2 -18817.353} C_VEL
LIN {X 0,Y 247.443,Z 305.821,A -85,B 0,C 180,E1 -18819.811,E2 -18819.811} C_VEL
LIN {X 0,Y 248.258,Z 299.287,A -85,B 0,C 180,E1 -18822.673,E2 -18822.673} C_VEL
LIN {X 0,Y 249.497,Z 292.122,A -85,B 0,C 180,E1 -18825.103,E2 -18825.103} C_VEL
LIN {X 0,Y 251.071,Z 283.177,A -85,B 0,C 180,E1 -18827.512,E2 -18827.512} C_VEL
LIN {X 0,Y 252.389,Z 273.966,A -85,B 0,C 180,E1 -18829.52,E2 -18829.52} C_VEL
LIN {X 0,Y 254.264,Z 263.817,A -85,B 0,C 180,E1 -18831.271,E2 -18831.271} C_VEL
LIN {X 0,Y 256.076,Z 252.518,A -85,B 0,C 180,E1 -18832.809,E2 -18832.809} C_VEL
LIN {X 0,Y 257.789,Z 239.808,A -85,B 0,C 180,E1 -18834.138,E2 -18834.138} C_VEL
LIN {X 0,Y 259.201,Z 227.408,A -85,B 0,C 180,E1 -18835.065,E2 -18835.065} C_VEL
LIN {X 0,Y 260.155,Z 213.716,A -85,B 0,C 180,E1 -18835.762,E2 -18835.762} C_VEL
LIN {X 0,Y 261.843,Z 154.835,A -85,B 0,C 180,E1 -18837.387,E2 -18837.387} C_VEL
LIN {X 0,Y 258.074,Z 124.183,A -85,B 0,C 180,E1 -18838.684,E2 -18838.684} C_VEL
LIN {X 0,Y 256.399,Z 113.487,A -85,B 0,C 180,E1 -18839.188,E2 -18839.188} C_VEL
LIN {X 0,Y 252.894,Z 103.87,A -85,B 0,C 180,E1 -18839.913,E2 -18839.913} C_VEL
LIN {X 0,Y 250.534,Z 92.371,A -85,B 0,C 180,E1 -18844.127,E2 -18844.127} C_VEL
LIN {X 0,Y 249.101,Z 86.462,A -85,B 0,C 180,E1 -18846.458,E2 -18846.458} C_VEL
LIN {X 0,Y 249.025,Z 86.466,A -85,B 0,C 180,E1 -18850.474,E2 -18850.474} C_VEL
LIN {X 0,Y 248.994,Z 86.469,A -85,B 0,C 180,E1 -18854.881,E2 -18854.881} C_VEL
LIN {X 0,Y 249.008,Z 86.469,A -85,B 0,C 180,E1 -18857.361,E2 -18857.361} C_VEL
LIN {X 0,Y 249.024,Z 86.448,A -85,B 0,C 180,E1 -18861.619,E2 -18861.619} C_VEL
LIN {X 0,Y 249.042,Z 86.462,A -85,B 0,C 180,E1 -18865.639,E2 -18865.639} C_VEL
LIN {X 0,Y 249.051,Z 86.462,A -85,B 0,C 180,E1 -18869.473,E2 -18869.473} C_VEL
LIN {X 0,Y 249.073,Z 86.453,A -85,B 0,C 180,E1 -18873.162,E2 -18873.162} C_VEL
LIN {X 0,Y 249.079,Z 86.46,A -85,B 0,C 180,E1 -18876.733,E2 -18876.733} C_VEL
LIN {X 0,Y 249.11,Z 86.444,A -85,B 0,C 180,E1 -18880.212,E2 -18880.212} C_VEL
LIN {X 0,Y 249.241,Z 86.436,A -85,B 0,C 180,E1 -18883.622,E2 -18883.622} C_VEL
LIN {X 0,Y 249.244,Z 86.429,A -85,B 0,C 180,E1 -18888.616,E2 -18888.616} C_VEL
LIN {X 0,Y 249.454,Z 86.411,A -85,B 0,C 180,E1 -18891.902,E2 -18891.902} C_VEL
LIN {X 0,Y 249.291,Z 86.423,A -85,B 0,C 180,E1 -18895.149,E2 -18895.149} C_VEL
LIN {X 0,Y 249.673,Z 86.382,A -85,B 0,C 180,E1 -18898.387,E2 -18898.387} C_VEL
LIN {X 0,Y 249.673,Z 86.383,A -85,B 0,C 180,E1 -18901.613,E2 -18901.613} C_VEL
LIN {X 0,Y 249.432,Z 86.409,A -85,B 0,C 180,E1 -18906.553,E2 -18906.553} C_VEL
LIN {X 0,Y 249.342,Z 86.425,A -85,B 0,C 180,E1 -18909.737,E2 -18909.737} C_VEL
LIN {X 0,Y 249.205,Z 86.434,A -85,B 0,C 180,E1 -18914.704,E2 -18914.704} C_VEL
LIN {X 0,Y 249.14,Z 86.448,A -85,B 0,C 180,E1 -18918.078,E2 -18918.078} C_VEL
LIN {X 0,Y 249.087,Z 86.447,A -85,B 0,C 180,E1 -18921.519,E2 -18921.519} C_VEL
LIN {X 0,Y 249.13,Z 86.452,A -85,B 0,C 180,E1 -18925.483,E2 -18925.483} C_VEL
LIN {X 0,Y 249.073,Z 86.459,A -85,B 0,C 180,E1 -18928.99,E2 -18928.99} C_VEL
LIN {X 0,Y 249.031,Z 86.463,A -85,B 0,C 180,E1 -18932.426,E2 -18932.426} C_VEL
LIN {X 0,Y 249.029,Z 86.464,A -85,B 0,C 180,E1 -18936.346,E2 -18936.346} C_VEL
LIN {X 0,Y 248.979,Z 86.472,A -85,B 0,C 180,E1 -18940.484,E2 -18940.484} C_VEL
LIN {X 0,Y 248.984,Z 86.471,A -85,B 0,C 180,E1 -18944.884,E2 -18944.884} C_VEL
LIN {X 0,Y 249.01,Z 86.465,A -85,B 0,C 180,E1 -18947.362,E2 -18947.362} C_VEL
LIN {X 0,Y 249.043,Z 86.465,A -85,B 0,C 180,E1 -18952.202,E2 -18952.202} C_VEL
LIN {X 0,Y 249.045,Z 86.462,A -85,B 0,C 180,E1 -18955.64,E2 -18955.64} C_VEL
LIN {X 0,Y 249.004,Z 86.466,A -85,B 0,C 180,E1 -18959.467,E2 -18959.467} C_VEL
LIN {X 0,Y 249.029,Z 86.464,A -85,B 0,C 180,E1 -18963.158,E2 -18963.158} C_VEL
LIN {X 0,Y 249.04,Z 86.579,A -85,B 0,C 180,E1 -18966.832,E2 -18966.832} C_VEL
LIN {X 0,Y 250.006,Z 89.286,A -85,B 0,C 180,E1 -18967.033,E2 -18967.033} C_VEL
LIN {X 0,Y 256.865,Z 103.155,A -85,B 0,C 180,E1 -18968.245,E2 -18968.245} C_VEL
LIN {X 0,Y 262.84,Z 119.558,A -85,B 0,C 180,E1 -18969.369,E2 -18969.369} C_VEL
LIN {X 0,Y 260.674,Z 191.621,A -85,B 0,C 180,E1 -18971.328,E2 -18971.328} C_VEL
LIN {X 0,Y 259.853,Z 205.405,A -85,B 0,C 180,E1 -18972.032,E2 -18972.032} C_VEL
LIN {X 0,Y 258.781,Z 218.275,A -85,B 0,C 180,E1 -18973.026,E2 -18973.026} C_VEL
LIN {X 0,Y 257.36,Z 230.763,A -85,B 0,C 180,E1 -18974.356,E2 -18974.356} C_VEL
LIN {X 0,Y 255.785,Z 241.896,A -85,B 0,C 180,E1 -18975.887,E2 -18975.887} C_VEL
LIN {X 0,Y 254.12,Z 251.935,A -85,B 0,C 180,E1 -18977.624,E2 -18977.624} C_VEL
LIN {X 0,Y 252.438,Z 260.996,A -85,B 0,C 180,E1 -18979.575,E2 -18979.575} C_VEL
LIN {X 0,Y 250.842,Z 269.817,A -85,B 0,C 180,E1 -18981.948,E2 -18981.948} C_VEL
LIN {X 0,Y 249.529,Z 276.919,A -85,B 0,C 180,E1 -18984.343,E2 -18984.343} C_VEL
LIN {X 0,Y 248.529,Z 282.583,A -85,B 0,C 180,E1 -18986.758,E2 -18986.758} C_VEL
LIN {X 0,Y 247.872,Z 287.047,A -85,B 0,C 180,E1 -18989.188,E2 -18989.188} C_VEL
LIN {X 0,Y 247.342,Z 290.457,A -85,B 0,C 180,E1 -18991.629,E2 -18991.629} C_VEL
LIN {X 0,Y 247.242,Z 292.147,A -85,B 0,C 180,E1 -18993.26,E2 -18993.26} C_VEL
LIN {X 0,Y 247.198,Z 293.932,A -85,B 0,C 180,E1 -18995.684,E2 -18995.684} C_VEL
LIN {X 0,Y 247.086,Z 294.859,A -85,B 0,C 180,E1 -18998.177,E2 -18998.177} C_VEL
LIN {X 0,Y 247.3,Z 294.652,A -85,B 0,C 180,E1 -19001.475,E2 -19001.475} C_VEL
LIN {X 0,Y 247.659,Z 293.968,A -85,B 0,C 180,E1 -19003.122,E2 -19003.122} C_VEL
LIN {X 0,Y 248.609,Z 291.734,A -85,B 0,C 180,E1 -19006.019,E2 -19006.019} C_VEL
LIN {X 0,Y 249.859,Z 288.187,A -85,B 0,C 180,E1 -19008.873,E2 -19008.873} C_VEL
LIN {X 0,Y 251.347,Z 283.976,A -85,B 0,C 180,E1 -19011.316,E2 -19011.316} C_VEL
LIN {X 0,Y 253.27,Z 278.284,A -85,B 0,C 180,E1 -19013.842,E2 -19013.842} C_VEL
LIN {X 0,Y 255.426,Z 271.734,A -85,B 0,C 180,E1 -19016.12,E2 -19016.12} C_VEL
LIN {X 0,Y 257.556,Z 264.744,A -85,B 0,C 180,E1 -19018.081,E2 -19018.081} C_VEL
LIN {X 0,Y 260.11,Z 255.569,A -85,B 0,C 180,E1 -19020.16,E2 -19020.16} C_VEL
LIN {X 0,Y 262.175,Z 246.968,A -85,B 0,C 180,E1 -19021.741,E2 -19021.741} C_VEL
LIN {X 0,Y 264.556,Z 236.784,A -85,B 0,C 180,E1 -19023.224,E2 -19023.224} C_VEL
